(* CODESYS project BaseVista.library
   Company: Vistaprint
   Title: Base_PLC
   Description: 0.3.5.10	- delete cmd on OFF/EOFF alarm
      	- delete SubState on state change
      	- alarm children propagation set true
      0.3.5.9	- goes to OFFBusy from EOFF
      	- added FurtherReactions to Always
      0.3.5.8 	- Added disable Child Alarm propagation functionality
      0.3.5.7 	- Added two actions to disable the EOFF and OFF Alarm transition
      0.3.5.6 	- fixed ERRORQuit
      0.3.5.5 	- TwinCAT 3.1 4016.12
      	- Added a Simulate all to the CIf.Info. This propagates the simulation comand down
      	- Added disable variables to the me for the EOff & Off Alarm and Comand
      	- Added new versions of Tc2_System & Tc2_Utilities
      0.3.5.4 	- added Full Name to CIf
      0.3.5.3 	- Compiled with 3.1 4016.6
      	- Added InstancePath to CIf.Info
      	- Added a property for InstancePath
      	- Fill CIf.Info.InstancePath in FB_init
      0.3.5.2 - CtrlInit() uses internal variable again, in cyclic call of FB at first caclic call and init not done - only init is executed
      	- Alarmhandler works now with time stamp FB, properties for timestamp usage in controller
      	- Add new functions strstr, initAllCtrl, callAllCtrlInit
      	- Integrate in BaseCtrl state logging
      	- Add logger system
      - Add time stamp FUB FB_TimeStamp
      0.3.5.1 - Add Methode ResetSubState
      - alarm reset first statemachine and then the messages
      0.3.5.0 - Update to TwinCat 4016.5
      0.3.4.9 - Increased maxchildnumber to 30
                  - CtrlInit made Public
                  - New CtrlInit call only once flag
      0.3.4.8 - BugFix setAlarm (rst,clr & set)
      0.3.4.7 - Increased the maxchildnumber to 25
      0.3.4.6 - Increased the maxchildnumber to 40
      0.3.4.5 - BugFix in alarm manager
      0.3.4.2 - Changed the Pramas Text in FB_CtrlBase
      0.3.4.1 - State single answer. Reset pending alarm class to NONE.
      0.3.4.0 - New CheckAllChildState also true feedback if check state of child OFF or EOFF and child in ERROR;
      - Bug fix Always Single-answer and startup with wait on PON
      - FB_Alm_Man: New Property IsInitDone		feedback at least one valid time stamp read out 
      0.3.3.7 - CheckParentAlmClass OFF and STOP added -> reaction of Controller
      0.3.3.6 - FB_Alm_Man Property CntPerClass added, alarm classes EOFF, OFF and STOP from parent to child, in EOFFBusy and OFF busy command in cyclic action (not entry action)
      
      0.3.3.4 - Added IO support for USINT datatype
      
      0.3.3.3 - Bug fixed in getInBolDebounced(FUN)
      
      0.3.3.2 - New function setAllCtrlAlarmFB -> all controller init pointer of alarmhandler; 
      - Rename GetInUint ->getInUint; 
      - New function ScaleINT (scale integer variable p.e. analog increment to 0.1mm)
      
      0.3.3.1  Added getInBolDebounced(FUN) and T_Ctrl_IoBoolDebounced(STRUCT) for debouncing inputs
      0.3.3.0 - Added pfbAlarmCtrl and the "zugehörige" property to allow clean alarm calls also from controllers in libraries.
      0.3.2.0 - Del getCtrlCIF,iniCtrlArray; Set cmds to child EOFF,OFF,PON; EOFF State; Check child ALM EOFF     
      0.3.1.3 - Bugfix
      0.3.1.2 - Added iniAllCtrlArrays - this is iniCtrlArray + the cif array
      0.3.1 - Added the automatic EOff propagation.
      0.3.0 - Added the substate to T_CTRL_CLASS_STATEMACHINE
      Automatic Substate handling.
      0.2.3 - Added support for sub usec cycletimes
      0.2.2 - Added the UInt for IO. T_CTRL_IOUint, setInUint(), setOutUint()
      0.2.1 - Added the property CtrlCIf to FB_CtrlBase
   Version: 0.3.5.10

Project tree, tasks and I/O mapping:
  libraries: Tc2_Standard, 3.3.0.0 (Beckhoff Automation GmbH); Tc2_System, 3.3.8.1 (Beckhoff Automation GmbH); Tc2_Utilities, 3.3.8.0 (Beckhoff Automation GmbH); Tc3_Interfaces, 3.3.0.0 (Beckhoff Automation GmbH); Tc3_MemMan, 3.3.1.0 (Beckhoff Automation GmbH); Tc3_Module, 3.3.6.0 (Beckhoff Automation GmbH)
  POUs/
    Alarm/
      data type E_AlmClass
      data type E_AlmCmd
      data type E_AlmState
      function block FB_Alm_Man [ST]: aCntPerClass, clearAlarm, IsInitDone, LocalTime_FileTime_BaseWin, LocalTime_TimeStruct_BaseWin, setAlarm, UTC_FileTime, UTC_TimeStruct
      data type T_AlmElement
      data type T_Ctrl_Alm
    BaseCtrl/
      global variables Base_CmdState
      global variables Base_Const
      data type E_Mode
      function block FB_CtrlBase [ST]: AddChild, AlarmCtrl, Always, BaseLog, CheckAllChildAlmClass, CheckAllChildState, CheckChildAlmClass, CheckCmdValid, CheckParentAlmClass, ChildrenAlarmPropagation, ClearAllSimulation, CtrlCIf, CtrlFB, CtrlInit, CycleEndDuty, CycleStartDuty, EOFF_EntryAction, EOffAlarmTransition, FB_init, FurtherReactions, getCmdState, iniAllCtrlArrays, InstancePath, IoInBridge, IoOutBridge, OffAlarmTransition, ResetSubState, SetAllChildAlmClass, SetAllChildCmd, SetAllSimulation, sta_EOFF, sta_EOFFBusy, sta_ERROR, sta_ERRORQuit, sta_OFF, sta_OFFBusy, sta_PON, sta_PONBusy, sta_SINGLE_ANSWER, StateMachine
      interface I_CtrlBase: CtrlCIf, CtrlFB
      data type T_Ctrl_AlarmConfig
      data type T_Ctrl_CIf
      data type T_Ctrl_Class
      data type T_Ctrl_Class_Alm
      data type T_Ctrl_Class_StateMachine
      data type T_Ctrl_CmdListElement
      data type T_Ctrl_Info
      data type T_Ctrl_IoBool
      data type T_Ctrl_IoBoolDebounced
      data type T_Ctrl_IoInt
      data type T_Ctrl_IoUint
      data type T_Ctrl_IoUsint
      data type T_Ctrl_Job
      data type T_Ctrl_SwCfg
      data type T_fbInfo
      data type T_StateLogger
    Utility/
      DLL (Double Linked List)/
        function block FB_DLL [ST]: addElement, deleteAll, deleteElement, FB_init, firstElement, numberOfElements, searchElement
        data type T_Element
      FileFolder/
        function block FB_FileCopy [ST]
        function block FB_FileHdl [ST]: ActFileSize, M_Cmd_FileDelete, M_Cmd_NewFile, M_Cmd_WriteBuffer, M_FileClose, M_FileCopy, M_FileDelete, M_FileOpen, M_FileRename, M_FileWrite, M_GetPathName, M_Init
        function block FB_FolderHdl [ST]: FileSupervisionPeriod, get_FileList, get_NewestFileEntry, M_Cmd_RefreshFileList, M_FileDelete, M_FileExist, M_getFileInfo, M_GetFileSize, M_Init, M_RefreshFileList, M_SortFileList, MaxNrOfFilesInFolder
        global variables FileHdl
      Logger/
        BasLog/
          global variables BasLog
          function block FB_BasLog [ST]: M_ChangeMask, M_CheckValidLogType, M_ClientInit, M_GetHandle, M_Log, M_Read
          function block FB_BasLogTest_Client [ST]
          function block FB_BasLogTest_Sender [ST]
          data type T_Bl_BaseStruc
          data type T_Bl_LibClient
          data type T_Bl_LibHandleRow
          data type T_Bl_LibSingleClient
        DatLog/
          global variables DatLog
          function block FB_DatLog [ST]: M_AllocMEM, M_CheckAndAppendDatLogInfo, M_GetHandle, M_Init, M_Log
          function block FB_DatLogTest_Sender [ST]
          data type T_DatLogTest
          data type T_DL_Item
          data type T_DL_LibInfo
          data type T_DL_Statemachine
          data type T_DL_SysInfo
        FileLc/
          function block FB_FileLc [ST]: M_Cyclic, M_Init, M_PutPvIdInList, M_ReleaseBuffer, M_WriteActItemIdx, M_WriteRecord
          function block FB_FileLc_FileHdl [ST]: ActFileSize, M_Cyclic, M_Init
          function block FB_FileLc_WorkOnFile [ST]: FB_exit, M_AllocMEM, M_ReleaseAllMEM
          function block FB_FileLcTest [ST]
          global variables FileLc
          data type T_FileLc_FileHandler
          data type T_FileLc_ItemCfg
          data type T_FileLc_ItemData
          data type T_FileLc_ItemInfo
          data type T_FileLc_LibInfo
          data type T_FileLc_RecordData
          data type T_FileLc_Statemachine
          data type T_FileLc_SysCfg
          data type T_FileLc_SysDebugInfo
          data type T_FileLc_SysInfo
      Queue/
        function block FB_Queue [ST]: FB_exit, M_AllocNewQueue, M_AllocNewQueueInfo, M_AllocNewQueueSystem, M_CheckAndAppendQueueSysInfo, M_Clear, M_GetHandle, M_GetHandle_TC, M_Init, M_Read, M_ReadReference, M_Write
        function block FB_QueueTest_Receiver [ST]
        function block FB_QueueTest_Sender [ST]
        global variables Queue
        data type T_Queue_Info
        data type T_Queue_InfoInternal
        data type T_Queue_LibInfo
        data type T_Queue_SysDebugInfo
        data type T_Queue_SysInfo
        data type T_Queue_TestData
      function callAllCtrlInit [ST]
      function block FB_TimeStamp [ST]: LocalTime_FileTime_BaseUTC, LocalTime_FileTime_BaseWin, LocalTime_TimeStruct_BaseUTC, LocalTime_TimeStruct_BaseWin, TimeZone_Refresh, UTC_FileTime, UTC_TimeStruct
      function getInBol [ST]
      function getInBolDebounced [ST]
      function getInInt [ST]
      function getInUint [ST]
      function getInUsint [ST]
      function getStrInstanceName [ST]
      function initAllCtrl [ST]
      function ScaleINT [ST]
      function setAllCtrlAlarmFB [ST]
      function setAllCtrlBasLogFB [ST]
      function setOutBol [ST]
      function setOutInt [ST]
      function setOutUint [ST]
      function setOutUsint [ST]
      function strstr [ST]
  Version/
    global variables Global_Version
*)

// POUs/Alarm/E_AlmClass
/// Do not change the sequence in this struct, such that the highest number is always the most important alarm!
TYPE E_AlmClass :
(
	///no alarm active
	NONE := 0,
	///info
	INFO,
	///warning
	WARNING,
	///tact stop
	TSTOP,
	///stop
	STOP,
	///off
	OFF,
	///Emergency off
	EOFF,
	Max_E_AlmClass
) INT;
END_TYPE

// POUs/Alarm/E_AlmCmd
TYPE E_AlmCmd :
(
	DONE := -1,
	INITIALIZED := 0,
	RESET_ALL := 2,
	RESET_RST := 4,
	RESET_CLR := 6,
	Max_E_AlmCmd
);
END_TYPE

// POUs/Alarm/E_AlmState
TYPE E_AlmState :
(
	///no alarm active
	NONE := 0,
	///alarm clear entry -> set bit1
	CLR := 1,
	///entry resettable alarm ->  set bit2
	RST := 2,
	///entry non resettable alarm ->  set bit2 + bit3
	SET := 3,
	Max_E_AlmState
);
END_TYPE

// POUs/Alarm/T_AlmElement
TYPE T_AlmElement :
STRUCT
	///unique alarm number := 100000*udiMachineNr + intCtrlId*100 + udiAlarmNr
	udiNr: UDINT;
	///additional information - better string???
	dinInfo: DINT;
	///corresponding alarm class
	eClass: E_AlmClass;
	///clear, resetable
	intState: E_AlmState;
	///entry time
	strDTEntry: STRING;
	///from machine (standard = 1)
	udiMachineNr: UDINT;
	///from controller
	intCtrlId: INT;
	///local alarm number
	udiAlarmNr: UDINT;
	// for debugging string alarm controller-alarm
	strText: STRING;
END_STRUCT
END_TYPE

// POUs/Alarm/T_Ctrl_Alm
TYPE T_Ctrl_Alm :
STRUCT
	///alarm flag array
	bol: BOOL;
	eAlmClass: E_AlmClass;
	strText: STRING;
END_STRUCT
END_TYPE

// POUs/BaseCtrl/E_Mode
{attribute 'qualified_only' := ''}
TYPE E_Mode :
(
	INITIALIZED := 0,
	AUTO := 10,
	SEMI := 11,
	MANU := 12
) INT;
END_TYPE

// POUs/BaseCtrl/T_Ctrl_AlarmConfig
TYPE T_Ctrl_AlarmConfig :
STRUCT
	// Disable the OFF Alarm transition
	bolOffAlarmTransitionDisable	: BOOL;
	// Disable the EOFF Alarm Transition
	bolEOffAlarmTransitionDisable	: BOOL;
	// Disable to Off Command Transition 
	bolOffCmdTransitionDisable		: BOOL;
	// Disable the EOffCommandTransition
	bolEOffCmdTransitionDisable		: BOOL;
	// Enable Alarm Propagation to Children
	bolChildrenAlarmPropagation		: BOOL;
END_STRUCT
END_TYPE

// POUs/BaseCtrl/T_Ctrl_CIf
TYPE T_Ctrl_CIf :
STRUCT
	Job: T_Ctrl_Job;
	Info: T_Ctrl_Info;
	SwCfg: T_Ctrl_SwCfg;
END_STRUCT
END_TYPE

// POUs/BaseCtrl/T_Ctrl_Class
TYPE T_Ctrl_Class :
STRUCT
	///local test flag to supress cyclic run (for debugging after init)
	bolActivate					: BOOL;
	intCmd						: INT;
	intCmdLast					: INT;
	eModeHistory				: E_Mode;
	///local flag mode change detected
	bolChangeBackToAUTO			: BOOL;
	StateMachine				: T_Ctrl_Class_StateMachine;
	SubStateMachine				: T_Ctrl_Class_StateMachine;
	Alarm						: T_Ctrl_Class_Alm;
	FUBInfo						: T_fbInfo;
	AlarmConfig					: T_Ctrl_AlarmConfig;
	// StateLogger infos
	stStateLogger : T_StateLogger;
	// Simulate All Executed
	bolSimulateAllExecuted			: BOOL;
END_STRUCT
END_TYPE

// POUs/BaseCtrl/T_Ctrl_Class_Alm
TYPE T_Ctrl_Class_Alm :
STRUCT
	bolResetOk: BOOL;
	///flag positive check me alarm from child
	bolfp: BOOL;
	///local activ alarm class of parent ctrl
	eParent_ActivAlmClass: E_AlmClass;
	///highest local activ alarm class
	eActivAlmClass: E_AlmClass;
END_STRUCT
END_TYPE

// POUs/BaseCtrl/T_Ctrl_Class_StateMachine
TYPE T_Ctrl_Class_StateMachine :
STRUCT
	///actual state
	intState: INT;
	///state of last cycle
	intStateLastCycle: INT;
	///save history backup p.e. in ERROR state
	intStateHistory: INT;
	///set state for next cycle
	intStateNext: INT;
	///[ms] to simulate state in SINGLE_ANSWER
	udiStateSimSetTime_ms: UDINT := 1000;
	///[ms] time in one state
	udiTimeInState_ms: UDINT;
	///[ms] time in one state
	relTimeInState_ms: REAL;
	///[us] time in one state
	udiTimeInState_us: UDINT;
END_STRUCT
END_TYPE

// POUs/BaseCtrl/T_Ctrl_CmdListElement
TYPE T_Ctrl_CmdListElement :
STRUCT
	///command implemented in controller
	intCmd: INT;
	///command is available info for UI
	bolAvailable: BOOL;
	/// Name of command. Important for UI.
	strName: STRING(80);
END_STRUCT
END_TYPE

// POUs/BaseCtrl/T_Ctrl_Info
TYPE T_Ctrl_Info :
STRUCT
	///name of controller instance
	strName				: STRING(80);
	///full name of controller instance
	strFullName			: STRING(80);
	///class of controller
	strType				: STRING(80);
	///unique controller instance identification number
	intCtrlId			: INT;
	///unique identification number of parent controller instance
	intParentCtrlId		: INT;
	///all inputs valid -> init done
	bolInitDone			: BOOL;
	///Childs
	p_afbChild			: ARRAY[0..Base_Const.cMaxNrOfChilds] OF POINTER TO FB_CtrlBase;
	///common interface array of childs
	p_aCIf				: ARRAY[0..Base_Const.cMaxNrOfChilds] OF POINTER TO T_Ctrl_CIf;
	// Child Count
	uinChildNbr			: UINT;
	// Absolut path to the controller
	strInstancePath		: STRING;
END_STRUCT
END_TYPE

// POUs/BaseCtrl/T_Ctrl_IoBool
TYPE T_Ctrl_IoBool :
STRUCT
	///mapped io variable to hardware
	map: BOOL;
	///shows the state of (input: mapped, output: set by programm respectiv at the moment one cycle later evtl. from the forcing if forcing active) -> necessary for what?
	state: BOOL;
	///variabel to/ from program
	intern: BOOL;
	///variabel set from UI
	force: BOOL;
	///enable force of single io-datapoint
	EnForce: BOOL;
END_STRUCT
END_TYPE

// POUs/BaseCtrl/T_Ctrl_IoBoolDebounced
TYPE T_Ctrl_IoBoolDebounced :
STRUCT
	///mapped io variable to hardware
	map: BOOL;
	///shows the state of (input: mapped, output: set by programm respectiv at the moment one cycle later evtl. from the forcing if forcing active) -> necessary for what?
	state: BOOL;
	///variabel to/ from program
	intern: BOOL;
	///variabel set from UI
	force: BOOL;
	///enable force of single io-datapoint
	EnForce: BOOL;
	// time since last input change
	udinDebouncedTimeCounter_ms: UDINT;
END_STRUCT
END_TYPE

// POUs/BaseCtrl/T_Ctrl_IoInt
TYPE T_Ctrl_IoInt :
STRUCT
	///mapped io variable to hardware
	map: INT;
	///shows the state of (input: mapped, output: set by programm respectiv at the moment one cycle later evtl. from the forcing if forcing active) -> necessary for what?
	state: INT;
	///variabel to/ from program
	intern: INT;
	///variabel set from UI
	force: INT;
	///enable force of single io-datapoint
	EnForce: BOOL;
END_STRUCT
END_TYPE

// POUs/BaseCtrl/T_Ctrl_IoUint
TYPE T_Ctrl_IoUint :
STRUCT
	///mapped io variable to hardware
	map: UINT;
	///shows the state of (input: mapped, output: set by programm respectiv at the moment one cycle later evtl. from the forcing if forcing active) -> necessary for what?
	state: UINT;
	///variabel to/ from program
	intern: UINT;
	///variabel set from UI
	force: UINT;
	///enable force of single io-datapoint
	EnForce: BOOL;
END_STRUCT
END_TYPE

// POUs/BaseCtrl/T_Ctrl_IoUsint
TYPE T_Ctrl_IoUsint :
STRUCT
	///mapped io variable to hardware
	map: USINT;
	///shows the state of (input: mapped, output: set by programm respectiv at the moment one cycle later evtl. from the forcing if forcing active) -> necessary for what?
	state: USINT;
	///variabel to/ from program
	intern: USINT;
	///variabel set from UI
	force: USINT;
	///enable force of single io-datapoint
	EnForce: BOOL;
END_STRUCT
END_TYPE

// POUs/BaseCtrl/T_Ctrl_Job
TYPE T_Ctrl_Job :
STRUCT
	///mode if mode = AUTO -> ACmd will be used, otherwise the MCmd channel is open
	eMode: E_Mode;
	///automatic command from parent ctrl
	intACmd: INT;
	///manual command from UI p.e.
	intMCmd: INT;
	///active cmd
	strCmd: STRING;
	///active state
	intState: INT;
	strState: STRING;
	///if used - show substates for debugging
	strSubState: STRING;
	///event channel to signal special events to parent parallel to status
	intEvt: INT;
	///reset all alarms
	bolAlmReset: BOOL;
	///activate io-forcing
	bolIoForce: BOOL;
	///overwrite suspend all interlocks (for debugging/testing)
	bolIlkOverwrite: BOOL;
	///activ alarm class of parent ctrl
	eParent_ActivAlmClass: E_AlmClass;
	///activ alarm class of me ctrl
	eMe_ActivAlmClass: E_AlmClass;
	///list of all implemented commands
	aCmdList: ARRAY[0..cMaxCmdPerCtrl] OF T_Ctrl_CmdListElement;
END_STRUCT
END_TYPE

// POUs/BaseCtrl/T_Ctrl_SwCfg
TYPE T_Ctrl_SwCfg :
	STRUCT
		///hardware/controller exists
		bolExist: BOOL;
		///enable statemachine
		bolEnable: BOOL;
		///set controller in simulation(statemachine active, io local simulated)
		bolSimulation: BOOL;
		//set controller and all sub controllers into simulation(statemachine active, io local simulated)
		bolAllSimulation: BOOL;
		// enable statelogger
		bolEnStateLogger: BOOL;
	END_STRUCT
END_TYPE

// POUs/BaseCtrl/T_fbInfo
TYPE T_fbInfo :
STRUCT
	bolCycleTimeBelowMS			: BOOL;
	udiSample_ms				: UDINT;
	udiSample_us				: UDINT;
END_STRUCT
END_TYPE

// POUs/BaseCtrl/T_StateLogger
TYPE T_StateLogger :
STRUCT
	pfbBaseLog : POINTER TO FB_BasLog; // should be set from outside over property
	uinStatus_Handle : UINT; // =0 handle ok or not allready requested 
	pHandle : POINTER TO T_Bl_LibHandleRow; // pointer to base logger system
	uinStatusWrite : UDINT; // feedback if write was successfully
	bolDoLog : BOOL; // state change detected or application cmd to log infos
	strText1: STRING(BasLog.cMAX_CHAR_TEXT1); // set in CycleEndDuty
	
	// free usable for application
	strText2: STRING(BasLog.cMAX_CHAR_TEXT2); // free usable from application task for additional debug informations
	dinPar3: DINT;	 // free usable from application task for additional debug informations
	dinPar4: DINT;	 // free usable from application task for additional debug informations
END_STRUCT
END_TYPE

// POUs/Utility/DLL (Double Linked List)/T_Element
{attribute 'enable_dynamic_creation' := ''}
TYPE T_Element :
STRUCT
	pPrevElement: POINTER TO T_Element;
	pData: POINTER TO BYTE;
	uliKey: ULINT;
	pNextElement: POINTER TO T_Element;
END_STRUCT
END_TYPE

// POUs/Utility/Logger/BasLog/T_Bl_BaseStruc
TYPE T_Bl_BaseStruc :
STRUCT
	dtDateTimeEntry: DT; // actual date and time (Date and time.The most significat digit is one second. 32Bit 1970-01-01-00:00 to 2106-02-06-06:28:15)
	uinMs : UINT; // actual millisecond
	udiLogType: UDINT; // kind of log
	intCtrlID: INT; // unique controllerID which element has created this entry
	strText1: STRING(BasLog.cMAX_CHAR_TEXT1);	//informationtext1
	strText2: STRING(BasLog.cMAX_CHAR_TEXT2); // informationtext2
	dinPar1: DINT; // value parmeter 1
	dinPar2: DINT; // value parmeter 2
	dinPar3: DINT; // value parmeter 3
	dinPar4: DINT; // value parmeter 4
END_STRUCT
END_TYPE

// POUs/Utility/Logger/BasLog/T_Bl_LibClient
TYPE T_Bl_LibClient :
STRUCT
	stClient : ARRAY [0..BasLog.cMAX_CLIENTS] OF T_Bl_LibSingleClient; // informationstruct for one client
	usiClientNr : USINT; // number of declared clients
	stHandleRow : ARRAY[0..Queue.cMAX_NR_OF_TASKS]OF T_Bl_LibHandleRow; // handle for access Buffer
	p_fbTimeStamp: POINTER TO FB_TimeStamp; // pointer to FB_TimeStamp 
END_STRUCT
END_TYPE

// POUs/Utility/Logger/BasLog/T_Bl_LibHandleRow
TYPE T_Bl_LibHandleRow :
STRUCT
	pQueueHandle :ARRAY[0..BasLog.cMAX_CLIENTS] OF POINTER TO T_Queue_Info; // handle for access buffer
	usiRequest: USINT; // information if task allready requested a handle
END_STRUCT
END_TYPE

// POUs/Utility/Logger/BasLog/T_Bl_LibSingleClient
TYPE T_Bl_LibSingleClient :
STRUCT
	strName : STRING(Queue.cMAX_NAME_LENGTH); // name of declared client
	udiMask : UDINT; // filter mask for selection
	udiNrOfElements: UDINT; // number of elements
	bolUseLocalTimeStamp : BOOL; // definition if using local time or UTC
END_STRUCT
END_TYPE

// POUs/Utility/Logger/DatLog/T_DatLogTest
TYPE T_DatLogTest :
STRUCT
	bolOk : BOOL := TRUE;
	intCnt : INT := 77;
	strNewText : STRING(20) := 'Test Data log';
END_STRUCT
END_TYPE

// POUs/Utility/Logger/DatLog/T_DL_Item
TYPE T_DL_Item :
STRUCT
	strPvName : T_MaxString; // name of declared client
	udiItemType : UDINT; // datatyp defined in logsystem
	uinItemOffset : UINT; // data offset in record struct
	SymInfo : SYMINFOSTRUCT;
END_STRUCT
END_TYPE

// POUs/Utility/Logger/DatLog/T_DL_LibInfo
TYPE T_DL_LibInfo :
STRUCT
	pstDatLogSysInfo : POINTER TO T_DL_SysInfo; // pointer to DL log system list
	stStatemachine: T_DL_Statemachine;
	udiCommonRecIdx: UDINT; // general record idx (because of mutex problematic has to be increased with 2)
END_STRUCT
END_TYPE

// POUs/Utility/Logger/DatLog/T_DL_Statemachine
TYPE T_DL_Statemachine :
STRUCT
	uinState : UINT; (*Status (Statemachine) des Filehandlers*)
	uinState_old : UINT; (*status old for entry action generation*)
	bolExecute_old : BOOL;
	usiInitDone : USINT; (*Merker für Neustart*)
END_STRUCT
END_TYPE

// POUs/Utility/Logger/DatLog/T_DL_SysInfo
TYPE T_DL_SysInfo :
STRUCT
	strDatLogName : STRING(DatLog.cMAX_SYS_NAME_LENGTH);
	usiInitOk : USINT; // initalisation successfully finished
	uinNbrOfItems : UINT; // number of items
	uinStartId : UINT; // StartId
	pBaseLogHandle : POINTER TO POINTER TO T_Queue_Info; // handle from BaseLog Init
	p_fbBasLog: POINTER TO FB_BasLog;
	pstItems: POINTER TO T_DL_Item; // itemlist
	uinCntReadItems : UINT; // read counte
	uinItemOffset : UINT; // offset calculation
	pstNextDatLogSystem : POINTER TO T_DL_SysInfo;
END_STRUCT
END_TYPE

// POUs/Utility/Logger/FileLc/T_FileLc_FileHandler
TYPE T_FileLc_FileHandler :
STRUCT
	uinState : UINT; (*Status (Statemachine) des Filehandlers*)
	uinState_old : UINT; (*status old for entry action generation*)
	usiCmd : USINT; (*Internes Kommando*)
	usiCmdNewFile : USINT; (*Schliesse aktuelles File ab und erstelle ein neues LogFile*)
	usiInitDone : USINT; (*Merker für Neustart*)
	udiWriteTimer : UDINT; (*Zeit seit letztem File Schreibzyklus*)
	p_bytTmpFileBuffer : POINTER TO BYTE; (*Zeiger auf temporären Filebuffer*)
	udiTmpFileBufferSize : UDINT; (*Grösse des temporären Filebuffers*)
	udiTmpFileBufferOffset : UDINT; (*Schreibzeiger des temporären Filebuffers*)
	udiRecordCnt : UDINT; // actual record count in file
	FB_FileLc_FileHdl : FB_FileLc_FileHdl; // FUB instance
	strInfo: Tc2_System.T_MaxString;	// additional debug Info
END_STRUCT
END_TYPE

// POUs/Utility/Logger/FileLc/T_FileLc_ItemCfg
TYPE T_FileLc_ItemCfg :
STRUCT
	dinPvId : DINT; (*Item - Id*)
	strPostText : STRING[FileLc.cPRE_POST_TEXTLEN]; (*Text, der nach dem Item - Value ins File geschrieben wird.*)
END_STRUCT
END_TYPE

// POUs/Utility/Logger/FileLc/T_FileLc_ItemData
TYPE T_FileLc_ItemData :
STRUCT
		udiRecIdx : UDINT; (*Record - Index, zu welchem die Daten gehören*)
		strValue : STRING[FileLc.cMAX_ITEM_CHAR]; (*Item - Value bereits in einen String gewandelt*)
END_STRUCT
END_TYPE

// POUs/Utility/Logger/FileLc/T_FileLc_ItemInfo
TYPE T_FileLc_ItemInfo :
STRUCT
	uinActNbrOfItems : UINT; (*Anzahl ermittelter Items*)
	strPreItemText : STRING[FileLc.cPRE_POST_TEXTLEN]; (*Text, der vor dem ersten Item - Value ins File geschrieben wird*)
	p_bytItemCfgList : POINTER TO T_FileLc_ItemCfg;; (*Zeiger auf die Item - Konfig - Liste*)
	stItemRecordData : ARRAY[0..Queue.cMAX_NR_OF_TASKS] OF T_FileLc_RecordData; (*Record - Data: Da Data - Records theoretisch unterbrochen werden können (Taskklassenprio), müssen mehrere Records quasi parallel behandelt werden können. Jeder Record hat daher seinen eigenen Index.*)
	a_p_bytItemDataList : ARRAY[0..Queue.cMAX_NR_OF_TASKS] OF POINTER TO BYTE; (*Item - Data: siehe oben...*)
END_STRUCT
END_TYPE

// POUs/Utility/Logger/FileLc/T_FileLc_LibInfo
TYPE T_FileLc_LibInfo :
STRUCT
	uinActNbrOfFileClients: UINT; // number of file clients
	uinActClientInitActive: UINT; // =0 ready for next client, actual active init of client nr
	stSysInfo : ARRAY[0..FileLc.cMAX_NBR_OF_FILECLIENTS] OF T_FileLc_SysInfo;
	p_fbBasLog: POINTER TO FB_BasLog; // only one central FB_BasLog instance allowed per PLC!!!
	fbTimeStamp: FB_TimeStamp; // only one central time for time stamps
END_STRUCT
END_TYPE

// POUs/Utility/Logger/FileLc/T_FileLc_RecordData
TYPE T_FileLc_RecordData :
STRUCT
	udiRecIdx : UDINT; (*Record - Index*)
	dtActDateTime : DATE_AND_TIME; (*Datum/Zeit der Record - Daten*)
	uinActMilli : UINT; (*Millisekunden der Record - Daten*)
END_STRUCT
END_TYPE

// POUs/Utility/Logger/FileLc/T_FileLc_Statemachine
TYPE T_FileLc_Statemachine :
STRUCT
	uinState : UINT; (*Status (Statemachine) des Filehandlers*)
	uinState_old : UINT; (*status old for entry action generation*)
	usiInitDone : USINT; (*Merker für Neustart*)
END_STRUCT
END_TYPE

// POUs/Utility/Logger/FileLc/T_FileLc_SysCfg
TYPE T_FileLc_SysCfg :
STRUCT
	uinMaxNbrOfLogFiles : UINT; (*Maximale Anzahl Log-Files*)
	udiTimeCheckMaxFileNr :UDINT; // [ms] time until check if more then max number of files exist in folder -> delete oldest
	uinNewFileOnRestart : UINT; (*Nach Steuerungsneustart neues File anlegen, wenn Wert > 0*)
	udiMaxTimeWriteToFile : UDINT; (*Maximale Zeit zwischen zwei File - Schreibzyklen*)
	bolUseLocalTimeStamp : BOOL; // define if using local time or UTC
	strLogFileNameExt : STRING[FileLc.cFILENAME_LENGTH]; (*Extension des Logfiles*)
	strLogFileNamePraeFix : STRING[FileLc.cFILENAME_LENGTH]; (*Präfix des Logfiles*)
	strLogPath : STRING[FileLc.cFILENAME_LENGTH]; (*Verzeichnis in welchem die Logfiles angelegt werden*)
	strLogNetId : STRING(23); // to access foreign system drives where TinCat has to be installed!!! Is a string containing the AMS network identifier of the target device to which the ADS command is directed.
	udiQueueLen : UDINT; (*Queue Länge der BaseLog - Queue*)
	udiMaxFileSize : UDINT; (*Maximale Dateigrösse eines Logfiles*)
	udiMaxEntriesInFile : UDINT; (*Maximale Anzahl Einträge in einem Logfile*)
END_STRUCT
END_TYPE

// POUs/Utility/Logger/FileLc/T_FileLc_SysDebugInfo
TYPE T_FileLc_SysDebugInfo :
STRUCT
		udiLogCounter : UDINT;
		uinGetHandleCalls : UINT;
END_STRUCT
END_TYPE

// POUs/Utility/Logger/FileLc/T_FileLc_SysInfo
TYPE T_FileLc_SysInfo :
STRUCT
	strPathName : STRING[FileLc.cPATH_LENGTH]; (*device name for config - file*)
	pBaseLogHandle : POINTER TO POINTER TO T_Queue_Info; // handle from BaseLog Init
	uinLogTyp : UINT; (* LogTyp*)
	udiMask : UDINT; (*actual log mask*)
	udiCylceTimeMs : UDINT; (*cycle time in milli seconds*)
	p_bytHeaderText : POINTER TO BYTE; (*Zeiger auf den Header Text*)
	udiHeaderTextLen : UDINT; (*Footer text len*)
	p_bytFooterText : POINTER TO BYTE; (*Zeiger auf den Footer Text*)
	udiFooterTextLen : UDINT; (*Footer text len*)
	p_bytTmpRecordText : POINTER TO BYTE; (*Zeiger auf den temporären Record - Text*)
	udiTmpRecordSize : UDINT; (*Grösse des temporären Record - Text*)
	udiTmpRecordLen : UDINT; (*Aktuelle Länge des temporären Record - Text*)
	bolTmpRecordFull : BOOL; (*temp record is full - text is full --> do write in file buffer*)
	stConfig : T_FileLc_SysCfg; (*config data*)
	stFileHandler : T_FileLc_FileHandler; (*Filehandler*)
	stItemInfo : T_FileLc_ItemInfo; (*Item-Infos --> <RECORD> Items.... </RECORD>*)
	stStatemachine : T_FileLc_Statemachine;
	fbFileLc_WorkOnFile : FB_FileLc_WorkOnFile;
END_STRUCT
END_TYPE

// POUs/Utility/Queue/T_Queue_Info
{attribute 'enable_dynamic_creation' := ''}
TYPE T_Queue_Info :
STRUCT
	fbBuffer: FB_MemRingBuffer; // Buffer FB
	udiFillLevel : UDINT; // % actual used buffer size
	pQueueSysInfo: POINTER TO T_Queue_SysInfo; // pointer to sytem struct (parent)
	bolAllocMe:BOOL; //flag gethandle called before init done!!!
END_STRUCT
END_TYPE

// POUs/Utility/Queue/T_Queue_InfoInternal
TYPE T_Queue_InfoInternal :
STRUCT
	bolAllocated:BOOL; //queue allocated
	fbBuffer: FB_MemRingBuffer; // Buffer FB
	udiFillLevel : UDINT; // % actual used buffer size
END_STRUCT
END_TYPE

// POUs/Utility/Queue/T_Queue_LibInfo
TYPE T_Queue_LibInfo :
STRUCT
	pstQueue_SysInfo : POINTER TO T_Queue_SysInfo; // pointer to first queue system - linked list 
	uinFUBInternalError: UINT; // internal error
	stSysDebugInfo:T_Queue_SysDebugInfo; //Debug structure
END_STRUCT
END_TYPE

// POUs/Utility/Queue/T_Queue_SysDebugInfo
TYPE T_Queue_SysDebugInfo :
STRUCT
	uinGetHandleCalls : UINT;
	uinIniCalls:UINT;
	uinCheckAndAppendQSCalls:UINT;
	uinAllocNewQSCalls: UINT;
	uinAllocNewQICalls: UINT;
	uinAllocnewQCalls:UINT;
END_STRUCT
END_TYPE

// POUs/Utility/Queue/T_Queue_SysInfo
{attribute 'enable_dynamic_creation' := ''}
TYPE T_Queue_SysInfo :
STRUCT
	strQueueName : STRING(Queue.cMAX_NAME_LENGTH); // queue name
	uinNbrOfElement : UINT; // number of elements
	udiSizeOfElement : UDINT; // Byte size of one elment
	uinMode : UINT; // 0: FIFO ring buffer, no overwrite!!
	// ident of FIFO new saved in fbBuffer udiIdent : UDINT;
	udiSecure: UDINT; // alternating bit muster for plausibility check of handle
	pQueueInfo: ARRAY[0..Queue.cMAX_NR_OF_TASKS] OF POINTER TO  T_Queue_Info; // structure/queue per tasclass
	pstNextQueue_SysInfo : POINTER TO T_Queue_SysInfo; // pointer to next queue system - linked list 
END_STRUCT
END_TYPE

// POUs/Utility/Queue/T_Queue_TestData
TYPE T_Queue_TestData :
STRUCT
	strName : STRING(34); //name OF process variabel
	usiDataTyp : USINT;
	udiDataLen : UDINT;
	udiDimension : UDINT;
	udiAdress : UDINT;
END_STRUCT
END_TYPE

// POUs/BaseCtrl/Base_CmdState
VAR_GLOBAL CONSTANT
	///ctrl commands definitions
	///general commands 2-200 - every command has to be a even number
	cCMD_DONE: INT := -1;
	cCMD_INITIALIZED: INT := 0;
	cCMD_PON: INT := 2;
	cCMD_EOFF: INT := 4;
	cCMD_OFF: INT := 6;
	cCMD_INIT: INT := 8;
	cCMD_RUN: INT := 10;
	cCMD_STOP: INT := 12;
	cCMD_TSTOP: INT := 14;
	///ctrl states definitions
	cSTA_DONE: INT := cCMD_DONE;
	cSTA_INITIALIZED: INT := cCMD_INITIALIZED;
	cSTA_PONBusy: INT := 1;
	cSTA_PON: INT := cCMD_PON;
	cSTA_EOFFBusy: INT := 3;
	cSTA_EOFF: INT := cCMD_EOFF;
	cSTA_OFFBusy: INT := 5;
	cSTA_OFF: INT := cCMD_OFF;
	cSTA_INITBusy: INT := 7;
	cSTA_INIT: INT := cCMD_INIT;
	cSTA_RUNBusy: INT := 9;
	cSTA_RUN: INT := cCMD_RUN;
	cSTA_STOPBusy: INT := 11;
	cSTA_STOP: INT := cCMD_STOP;
	cSTA_TSTOPBusy: INT := 13;
	cSTA_TSTOP: INT := cCMD_TSTOP;
	///special states without corresponding cmd
	cSTA_ERROR: INT := 150;
	cSTA_ERRORQuit: INT := 151;
	cSTA_SINGLE_ANSWER: INT := 152;
END_VAR

// POUs/BaseCtrl/Base_Const
VAR_GLOBAL CONSTANT
	///number of child access possible in one controller class
	cMaxNrOfChilds: UINT := 30;
	///maximal number of commands implemented in one controller class
	cMaxCmdPerCtrl: UINT := 15;
	///maximal number of commands implemented in one controller class
	cMaxBaseCmdState: UINT := 200;
END_VAR

// POUs/Utility/FileFolder/FileHdl
VAR_GLOBAL CONSTANT
	cFILE_HDL_MAX_NR_OF_FILE_TO_MANAGE: UDINT := 500;
END_VAR

// POUs/Utility/Logger/BasLog/BasLog
VAR_GLOBAL CONSTANT
	// internal
	cCLIENT_NAME_PF : STRING(10) := '__logClnt'; //Prefix for client name
	cVAR_TYPE_CMD_NEW_REC : USINT := 201; // command for log-records (collect multiple base log entries)
	cVAR_TYPE_CMD_END_REC : USINT := 202; // command for log-records (collect multiple base log entries)
	
	// limits
	cMAX_CLIENTS : USINT := 5; // maximal number of clients 
	cMAX_CHAR_TEXT1: USINT := 80;	// maximal number of chars for information text1
	cMAX_CHAR_TEXT2: USINT := 80;	// maximal number of chars for information text2	
	
	// log types
	cLOGTYPE_ALARM : UDINT:=1; //logtyp alarm
	cLOGTYPE_WARNING : UDINT:=2; //logtyp warning
	cLOGTYPE_INFO : UDINT:=4; //logtyp info
	cLOGTYPE_STATELOG : UDINT:=8; //logtyp state log (for statmachine diagnostic)
	cLOGTYPE_PV_EVENT : UDINT:=16; //logtyp triggered value log
	cLOGTYPE_PV_CYCLIC : UDINT:=32; //logtyp cyclic value log 
	cLOGTYPE_DATA : UDINT:=64; //logtyp data logger
	
	// error number
	cERR_TOO_MANY_CLIENTS : UINT := 51001; // max number of clients connected
	cERR_SYSTEM_NOT_FOUND : UINT := 51002; // the system with this name does not exist
	cERR_INVALID_LOGTYPE : UINT := 51003; // log type is not correct bit coded
	cERR_NO_WRITE_TASK : UINT := 51004; // no client added (no handle from a task)
	cERR_NO_HANDLE : UINT := 51005; // no handle received => fbGetHandle()
	cERR_NO_FB_TIME_STAMP_POINTER : UINT := 51006; // no pointer for FB_TimeStamp
	cERR_NO_FB_TIME_STAMP_INIT_NOT_OK : UINT := 51007; // time stamp value not ready for read out
END_VAR

// POUs/Utility/Logger/DatLog/DatLog
VAR_GLOBAL CONSTANT
	// internal
	cVAR_TYPE_BOOL : USINT := 1; (*Variable hat den Datentyp BOOL*)
	cVAR_TYPE_SINT : USINT := 2; (*Variable hat den Datentyp SINT*)
	cVAR_TYPE_INT : USINT := 3; (*Variable hat den Datentyp INT*)
	cVAR_TYPE_DINT : USINT := 4; (*Variable hat den Datentyp DINT*)
	cVAR_TYPE_USINT : USINT := 5; (*Variable hat den Datentyp USINT*)
	cVAR_TYPE_UINT : USINT := 6; (*Variable hat den Datentyp UINT*)
	cVAR_TYPE_UDINT : USINT := 7; (*Variable hat den Datentyp UDINT*)
	cVAR_TYPE_LREAL : USINT := 10; (*Variable hat den Datentyp REAL*)
	cVAR_TYPE_REAL : USINT := 8; (*Variable hat den Datentyp REAL*)
	cVAR_TYPE_STRING : USINT := 9; (*Variable hat den Datentyp STRING*)
	cVAR_TYPE_DATE_AND_TIME : USINT := 11; (*Variable hat den Datentyp DATE_AND_TIME*)
	cCTRL_ID : INT := 32001; // control ID from data log

	// limits	
	cMAX_SYS_NAME_LENGTH : USINT := 30; //max name length of system data log name
	cMAX_VAR_NAME_LEN : USINT := 50; // max len of variable name
	cMAX_NR_OF_VAR : UINT := 20; // max number of variables definable to log

	// error number	
	cERR_MEM_ALLOC : UINT := 53001; // error on allocating memory 
	cERR_NO_HANDLE : UINT := 53002; // no handle received => fbGetHandle()
	cERR_NO_DATE : UINT := 53003; // no valid data pointer received
	cERR_INIT_FAILED : UINT := 53006; // 
	cERR_NO_ITEMS : UINT := 53004; // 
	cERR_UNSUPPORTED_TYPE : UINT := 53005; // the system support this datatyp not
	cERR_UNSUPPORTED_TYPE_STRING_TOO_LONG : UINT := 53006; // defined string in base log shorter then log string
END_VAR

// POUs/Utility/Logger/FileLc/FileLc
VAR_GLOBAL CONSTANT
	// internal
	cVAR_TYPE_BOOL : USINT := 1; (*Variable hat den Datentyp BOOL*)
	cVAR_TYPE_SINT : USINT := 2; (*Variable hat den Datentyp SINT*)
	cVAR_TYPE_INT : USINT := 3; (*Variable hat den Datentyp INT*)
	cVAR_TYPE_DINT : USINT := 4; (*Variable hat den Datentyp DINT*)
	cVAR_TYPE_USINT : USINT := 5; (*Variable hat den Datentyp USINT*)
	cVAR_TYPE_UINT : USINT := 6; (*Variable hat den Datentyp UINT*)
	cVAR_TYPE_UDINT : USINT := 7; (*Variable hat den Datentyp UDINT*)
	cVAR_TYPE_LREAL : USINT := 10; (*Variable hat den Datentyp REAL*)
	cVAR_TYPE_REAL : USINT := 8; (*Variable hat den Datentyp REAL*)
	cVAR_TYPE_STRING : USINT := 9; (*Variable hat den Datentyp STRING*)
	cVAR_TYPE_DATE_AND_TIME : USINT := 11; (*Variable hat den Datentyp DATE_AND_TIME*)
	
	// config file
	cTAG_TEMPLATE_E : STRING[80] := '</TEMPLATE>'; (*End Tag*)
	cTAG_TEMPLATE_B : STRING[80] := '<TEMPLATE>'; (*Start Tag*)
	cTAG_ROW_E : STRING[80] := '</ROW>'; (*End Tag*)
	cTAG_ROW_B : STRING[80] := '<ROW>'; (*Start Tag*)
	cTAG_RECORD_E : STRING[80] := '</RECORD>'; (*End Tag*)
	cTAG_RECORD_B : STRING[80] := '<RECORD>'; (*Start Tag*)
	cTAG_ITEM_E : STRING[80] := '</ITEM>'; (*End Tag*)
	cTAG_ITEM_B : STRING[80] := '<ITEM>'; (*Start Tag*)
	cTAG_HEADER_E : STRING[80] := '</HEADER>'; (*End Tag*)
	cTAG_HEADER_B : STRING[80] := '<HEADER>'; (*Start Tag*)
	cTAG_FOOTER_E : STRING[80] := '</FOOTER>'; (*End Tag*)
	cTAG_FOOTER_B : STRING[80] := '<FOOTER>'; (*Start Tag*)
	cTAG_CONFIG_E : STRING[80] := '</CONFIG>'; (*End Tag*)
	cTAG_CONFIG_B : STRING[80] := '<CONFIG>'; (*Start Tag*)
	
	// config tags
	cTAG_CFG_LOGFILE_PRAEFIX_E : STRING[80] := '</LOGFILE_PRAEFIX>'; (*End Tag*)
	cTAG_CFG_LOGFILE_PRAEFIX_B : STRING[80] := '<LOGFILE_PRAEFIX>'; (*Start Tag*)
	cTAG_CFG_LOGFILE_EXT_E : STRING[80] := '</LOGFILE_EXT>'; (*End Tag*)
	cTAG_CFG_LOGFILE_EXT_B : STRING[80] := '<LOGFILE_EXT>'; (*Start Tag*)
	cTAG_CFG_QUEUE_LEN_E : STRING[80] := '</QUEUE_LEN>'; (*End Tag*)
	cTAG_CFG_QUEUE_LEN_B : STRING[80] := '<QUEUE_LEN>'; (*Start Tag*)
	cTAG_CFG_LOGTYPE_E : STRING[80] := '</LOG_TYPE>'; (*End Tag*)
	cTAG_CFG_LOGTYPE_B : STRING[80] := '<LOG_TYPE>'; (*Start Tag*)
	cTAG_CFG_MASK_E : STRING[80] := '</LOG_MASK>'; (*End Tag*)
	cTAG_CFG_MASK_B : STRING[80] := '<LOG_MASK>'; (*Start Tag*)
	cTAG_CFG_MAX_LOGFILES_E : STRING[80] := '</MAX_LOGFILES>'; (*End Tag*)
	cTAG_CFG_MAX_LOGFILES_B : STRING[80] := '<MAX_LOGFILES>'; (*Start Tag*)
	cTAG_CFG_T_CHECK_MAX_FILE_NR_E : STRING[80] := '</TIME_CHECK_MAX_FILE_NR>'; (*End Tag*)
	cTAG_CFG_T_CHECK_MAX_FILE_NR_B : STRING[80] := '<TIME_CHECK_MAX_FILE_NR>'; (*Start Tag*)
	cTAG_CFG_MAX_T_TO_WRITE_E : STRING[80] := '</MAX_TIME_TO_WRITE>'; (*End Tag*)
	cTAG_CFG_MAX_T_TO_WRITE_B : STRING[80] := '<MAX_TIME_TO_WRITE>'; (*Start Tag*)
	cTAG_CFG_NEW_FILE_RESTART_E : STRING[80] := '</NEW_FILE_ON_RESTART>'; (*End Tag*)
	cTAG_CFG_NEW_FILE_RESTART_B : STRING[80] := '<NEW_FILE_ON_RESTART>'; (*Start Tag*)
	cTAG_CFG_MAX_ENTR_IN_FILE_E : STRING[80] := '</MAX_ENTRIES_IN_FILE>'; (*End Tag*)
	cTAG_CFG_MAX_ENTR_IN_FILE_B : STRING[80] := '<MAX_ENTRIES_IN_FILE>'; (*Start Tag*)
	cTAG_CFG_MAX_FILE_SIZE_E : STRING[80] := '</MAX_FILE_SIZE>'; (*End Tag*)
	cTAG_CFG_MAX_FILE_SIZE_B : STRING[80] := '<MAX_FILE_SIZE>'; (*Start Tag*)
	cTAG_CFG_LOG_TIMESTAMP_E : STRING[80] := '</LOG_TIMESTAMP>'; (*End Tag*)
	cTAG_CFG_LOG_TIMESTAMP_B : STRING[80] := '<LOG_TIMESTAMP>'; (*Start Tag*)
	cTAG_CFG_LOGFILE_SNETID_E : STRING[80] := '</LOGFILE_SNETID>'; (*End Tag*)
	cTAG_CFG_LOGFILE_SNETID_B : STRING[80] := '<LOGFILE_SNETID>'; (*Start Tag*)
	cTAG_CFG_LOGFILE_PATH_E : STRING[80] := '</LOGFILE_PATH>'; (*End Tag*)
	cTAG_CFG_LOGFILE_PATH_B : STRING[80] := '<LOGFILE_PATH>'; (*Start Tag*)
	cLOG_TIMESTAMP_WIN : STRING[80] := 'LOCAL_TIME'; (*using local time (windows time with time zone)*)
	cLOG_TIMESTAMP_UTC : STRING[80] := 'UTC'; (*using UTC*)
	
	//<ITEM>***</ITEM> predefined items of base log
	cITEM_UNIX_DATE_TIME_STR : STRING[80] := 'DT_UNIX_STR'; (*Item UNIX Datum/Zeit als String*)
	cITEM_UNIX_DATE_TIME : STRING[80] := 'DT_UNIX'; (*Item UNIX Datum/Zeit als Integer*)
	cITEM_TIME_MILLI : STRING[80] := 'TIME_MILLI'; (*Item Millisekunden*)
	cITEM_EXCEL_DATE_TIME : STRING[80] := 'DT_EXCEL'; (*Item date/time in Excel format. Days as real since 1.1.1980*)
	cITEM_DATE_SLASH_TIME_COLON : STRING[80] := 'DATE_SLASH_TIME_COLON'; //english date format 2014/09/23 07:10:24
	cITEM_BL_LOGTYP : STRING[80] := 'BL_LOGTYP'; (*Base Log Item LogTyp*)
	cITEM_BL_CTRL_ID : STRING[80] := 'BL_CTRL_ID'; (*Base Log Item Controller Id*)
	cITEM_BL_STRING1 : STRING[80] := 'BL_STRING1'; (*Base Log Item STRING 1*)
	cITEM_BL_STRING2 : STRING[80] := 'BL_STRING2'; (*Base Log Item STRING 2*)
	cITEM_BL_PAR1 : STRING[80] := 'BL_PAR1'; (*Base Log Item PAR1  *)
	cITEM_BL_PAR2 : STRING[80] := 'BL_PAR2'; (*Base Log Item PAR2*)
	cITEM_BL_PAR3 : STRING[80] := 'BL_PAR3'; (*Base Log Item PAR3*)
	cITEM_BL_PAR4 : STRING[80] := 'BL_PAR4'; (*Base Log Item PAR4*)
	
	// <LOG_TYPE>****</LOG_TYPE>	 predefined values
	cLOGTYP_BL_STR : STRING[80] := 'BL'; (*BaseLog*)
	cLOGTYP_PV_STR : STRING[80] := 'PV'; (*PVLog*)
	cLOGTYP_DATA_STR : STRING[80] := 'DATA'; (*DataLog*)
	cLOGTYP_OPEN_STR : STRING[80] := 'OPEN'; (*Item date/time in Excel format. Days as real since 1.1.1970*)
	
	// Defaults
	cLOGTYP_BL : USINT := 1; (*Baselog*)
	cLOGTYP_PV : USINT := 2; (*PV*)
	cLOGTYP_DATA : USINT := 3; (*Data*)
	cLOGTYP_OPEN : USINT := 4; (*Open --> Maske setzen!*)
	cPVTYPE_UNIX_DATE_TIME_STR : DINT := -3;
	cPVTYPE_UNIX_DATE_TIME : DINT := -1;
	cPVTYPE_DATE_SLASH_TIME_COLON : DINT := -13; //english date format 2014/09/23 07:10:24
	cPVTYPE_TIME_MILLI : DINT := -2;
	cPVTYPE_EXCEL_DATE_TIME : DINT := -4;
	cPVTYPE_BL_LOGTYP : DINT := -5;
	cPVTYPE_BL_CTRL_ID : DINT := -6;
	cPVTYPE_BL_STRING1 : DINT := -7;
	cPVTYPE_BL_STRING2 : DINT := -8;
	cPVTYPE_BL_PAR1 : DINT := -9;
	cPVTYPE_BL_PAR2 : DINT := -10;
	cPVTYPE_BL_PAR3 : DINT := -11;
	cPVTYPE_BL_PAR4 : DINT := -12;
	cTIME_CHECK_MAX_FILE_NR : UDINT := 300; //[s] time period until check number of files in folder
	cMAX_ITEM_CHAR : UINT := BasLog.cMAX_CHAR_TEXT1; (*25 ist das absolute Minimum für DATE_AND_TIME - String Darstellung*)
	cEOL : ARRAY[0..1] OF BYTE := [13,10]; (*End of Line (Line feed, carriage return)*)
	cCMD_FLUSHBUF_NEWFILE : USINT := 2;
	cCMD_FLUSHBUF : USINT := 1;
	cCFG_TIME_WRITE_TO_FILE : UDINT := 60; (*DEFAULT: Mindestens alle 60 Sekunden ins File schreiben*)
	cCFG_QUEUE_LEN : UDINT := 512; (*DEFAULT: Anzahl Elemente der Log Queue*)
	cCFG_LOGFILE_NAME : STRING[80] := 'LogData_'; (*DEFAULT: LogFile Präfix*)
	cCFG_LOGFILE_EXT : STRING[80] := 'txt'; (*DEFAULT: LogFile Extension*)
	cCFG_DEFAULT_MASK : UDINT := 16#FFFFFFFF; // Default mask
	cCFG_MAX_NBR_OF_LOGFILES : UINT := 2; // Defaultmax number of log files
	
	// limits
	cPRE_POST_TEXTLEN : UINT := 256; // max text len for pre and post text of a value
	cMAX_RECORDS_IN_FILE_BUF : UINT := 4; (*factor for calculation of file buffer*)
	cMAX_NBR_OF_FILECLIENTS : UINT := 10; (*Max number of file clients*)
	cFILENAME_LENGTH : UINT := 260; // config file name len
	cPATH_LENGTH : UINT := 260; // folderpath string len
	
	// error number	
	cERR_NBR_OF_FC_EXEEDED : UINT := 50400; (*Max number of file clients reached*)
	cERR_FILENAME_MISSING : UINT := 50401; (*Filename missing*)
	cERR_PATH_MISSING : UINT := 50402; (*Path definition missing*)
	cERR_CONFIG_TAG : UINT := 50403; (*Error in <CONFIG></CONFIG> tag*)
	cERR_TEMPLATE_TAG : UINT := 50404; (*Error in <TEMPLATE></TEMPLATE> tag*)
	cERR_INVALID_LOGTYP : UINT := 50405; (*Unknown or missing log type -> template/config - file*)
	cERR_HEADER_TAG : UINT := 50406; (*Error in <HEADER></HEADER> tag*)
	cERR_RECORD_TAG : UINT := 50407; (*Error in <RECORD></RECORD> tag*)
	cERR_ROW_TAG : UINT := 50408; (*Error in <ROW></ROW> tag*)
	cERR_ITEM_TAG : UINT := 50409; (*Error in <ITEM></ITEM> tag*)
	cERR_FOOTER_TAG : UINT := 50410; (*Error in <FOOTER></FOOTER> tag*)
	cERR_HANDLE : UINT := 50411; (*no handle reached*)
	cERR_INVALID_DEVICE : UINT := 50412; (*File destination not correct*)
	cERR_ALLOC_BUFFER_FILE_CONFIG : UINT := 50413; (*No memory available for config read out*)
	cERR_ALLOC_MEMORY : UINT := 50414; (*No memory available*)
	cERR_NO_BASELOG : UINT := 50415; (*BaseLog pointer invalid*)
	cERR_NO_FLCIDX : UINT := 50416; (*INIT not possibel no valid act client nr index reference / pointer invalid*)
END_VAR

// POUs/Utility/Queue/Queue
VAR_GLOBAL CONSTANT
	// internal
	cSECURE_CODE: UDINT := 1431655765; // alternating bit muster 0x55555555 -> for validation of queues
	
	// limits
	cMAX_NAME_LENGTH : UINT := 80; // maximal string length of queue name
	cMAX_NR_OF_TASKS: USINT := 6; // for the moment enough

	// error number
	cERR_QUEUE_FULL : UINT := 1; 
	cERR_QUEUE_EMPTY : UINT := 2; 
	cERR_QUEUE_NAME : UINT := 50000; // not valid or empty queue name
	cERR_NR_OF_ELEMENTS : UINT := 50001; // number of elements =0 
	cERR_SIZE_OF_ELEMENTS: UINT := 50002; // element size =0
	cERR_MEM_ALLOC  : UINT := 50003; // error allocate memory
	cERR_QUEUE_DOES_NOT_EXIST : UINT := 50004; // queue does not exist
	cERR_Q_INFO_DOES_NOT_EXIST : UINT := 50005; // queue info does not exist
	cERR_DATA_INVALID : UINT := 50006; // pointer to data not valid
	cERR_HANDLE_INVALID : UINT := 50007; // handle not ok
	cERR_TC_INVALID : UINT := 50008; // task class index not ok
	cERR_CLEAR : UINT := 50009; // clear of queue not ok
END_VAR

// Version/Global_Version
// This function has been automatically generated from the project information.
VAR_GLOBAL CONSTANT
	{attribute 'const_non_replaced'}
	stLibVersion_Base_PLC : ST_LibVersion := (iMajor := 0, iMinor := 3, iBuild := 5, iRevision := 10, sVersion := '0.3.5.10');
END_VAR

// POUs/Alarm/FB_Alm_Man
FUNCTION_BLOCK FB_Alm_Man
VAR_INPUT
	;
END_VAR
VAR_IN_OUT
	bolCtrlRst: BOOL; // reset all controller
END_VAR

VAR CONSTANT
	/// config alarm handler number of elements of queue
	c_uinMaxAlmElements: UINT := 99;
	/// 0: with history on PLC, auto clr alarms from array if alarm state clear is set
	c_uinModeAlarm: UINT := 1;
	/// machine number 1, at the moment every time set to 1
	c_udiMachineNr: UDINT := 1;
	/// commands from the UI
	cCMD_RESET_ALL: INT := 2;
	/// reset state=RST, reset state CLR
	cCMD_RESET_RST: INT := 4;
	/// reset state CLR -> c_uinModeAlarm = 1, automatic reset will be done on PLC
	cCMD_RESET_CLR: INT := 6;
END_VAR
VAR
	///------------------------------------------------------------
	/// UI interface
	/// alarmarray PLC -> UI
	aAlm: ARRAY[0..c_uinMaxAlmElements] OF T_AlmElement;
	/// command interface for UI -> PLC
	intAlmCmd: INT;
	///------------------------------------------------------------
	fbTimeStamp: FB_TimeStamp; // only one central time for time stamps

	jj: UINT;
	EmptyAlmElement: T_AlmElement;
	intState: INT;
	intTestCtrl: INT := 12;
	intTestState: INT;
	udiTestAlarmNr: UDINT;
	dinTestInfo: DINT;
	aCtrlAlm: ARRAY[1..6] OF T_Ctrl_Alm;
	eActiveAlmClass: E_AlmClass;

	aCntActiveAlmPerClass: ARRAY[0..(E_AlmClass.Max_E_AlmClass-1)] OF UINT; // count off all active alarms per class, idx=0 all active alarms
END_VAR

(*__________________________________________________________________________________________________
¦	
¦	Vistaprint Schweiz GmbH
¦	CH - 8401 Winterthur
¦
¦	www.vistaprint.ch - info@vistaprint.ch
¦___________________________________________________________________________________________________

Function desription:
The alarm manager sets and clears alarms from the internal array. In the internal array all active 
alarms of a machine are listed. The list has no order. A new entry will be inserted at the next 
free place.

For the easy usage for UI the function block is to be define as global. And then the cmd for reset should be 
set when the button is pressed -> intAlmCmd = cCMD_RESET_ALL
All active alarms are shown in the aAlm array.

History:
Version		Date			Author		Comment
---------------------------------------------------------------------------------------------------
0.00.1		29.04.2013		AVME/KVO	Start history
0.00.2		06.01.2014		AVME/PRE	Implement the counted active messages array
0.00.3		17.02.2014		AVME/KVO	New Property IsInitDone 
										feedback at least one valid time stamp read out 
										-> check at startup before cyclic call of FB's to avoid alarms without valid timestamp
0.00.4		16.05.2014		AVME/DSC	-> Inserted new "setAlarm" Method from Patrik C. (code review)									
										-> BugFix, build sum of all active alarms
0.00.5		07.07.2014		AVME/KVO	-> BugFix Method setAlarm , clr and reset -> also possibel if one entry is zero possibel
0.00.6		07.10.2014		AVME/KVO	-> BugFix alarm reset first statemachine and then the messages	
0.00.7		27.10.2014		AVME/KVO	-> delete GETSYSTEMTIME use FB_TimeStamp
										-> New time properties for easy access of every controller if needed
___________________________________________________________________________________________________*)

// call time stamp asynchronous synchronisation
fbTimeStamp.In_strNetId := ''; // use system time of log target system
fbTimeStamp.In_t_CycleTimeRefreshTimeZone := T#0S; // cyclic check time zone settings - not needed using LocalTime_FileTime_BaseWin for log system and local time
fbTimeStamp();

// interface for UI access
CASE intState OF
		
	0: // reset cmd
		intAlmCmd := cCMD_DONE; // Ready for new cmd
		intState := intState + 1;
		
	1: // wait for cmd
		IF (intAlmCmd=cCMD_RESET_ALL) OR (intAlmCmd=cCMD_RESET_CLR) OR  (intAlmCmd=cCMD_RESET_RST) THEN
			intState := intState + 1;
		END_IF
		
	2: // firt reset state machines -> leave Error state
		bolCtrlRst := TRUE;
		intState := intState + 1;
		
	3: // reset alarms / messages
		// reset state=RST, reset state CLR
		THIS^.clearAlarm(((intAlmCmd=cCMD_RESET_ALL) OR (intAlmCmd=cCMD_RESET_RST)), TRUE);
		intState := intState + 1;
		
	4: 
		intState := 0; // done
END_CASE

// build sum of all active alarms
aCntActiveAlmPerClass[0] := 0;
FOR jj:= 1 TO INT_TO_UINT(E_AlmClass.Max_E_AlmClass-1) BY 1 DO
	aCntActiveAlmPerClass[0] := aCntActiveAlmPerClass[0] + aCntActiveAlmPerClass[jj];
END_FOR

//**********************************************************************************************
// Test manual set/reset/clear alarm
//**********************************************************************************************
CASE intTestState OF
	
	0: // wait
		
	1: //CLR
		THIS^.setAlarm(intTestCtrl,udiTestAlarmNr,dinTestInfo,ADR(aCtrlAlm),E_AlmState.CLR,eActiveAlmClass);
		intTestState := 0;
		
	2: // RST
		THIS^.setAlarm(intTestCtrl,udiTestAlarmNr,dinTestInfo,ADR(aCtrlAlm),E_AlmState.RST,eActiveAlmClass);
		intTestState := 0;
		
	3: // SET
		THIS^.setAlarm(intTestCtrl,udiTestAlarmNr,dinTestInfo,ADR(aCtrlAlm),E_AlmState.SET,eActiveAlmClass);
		intTestState := 0;

END_CASE

PROPERTY PUBLIC aCntPerClass : ARRAY[0..(E_AlmClass.Max_E_AlmClass-1)] OF UINT
GET
aCntPerClass := aCntActiveAlmPerClass;
END_GET
END_PROPERTY

METHOD clearAlarm : BOOL
VAR_INPUT
	///-> clear all entries with state RST
	bolClear_RST: BOOL;
	///-> clear all entries with state CLR
	bolClear_CLR: BOOL;
END_VAR
VAR
	ii: UINT;
END_VAR
FOR ii:= 0 TO INT_TO_UINT(E_AlmClass.Max_E_AlmClass-1) BY 1 DO
	aCntActiveAlmPerClass[ii] := 0; // reset alarm counter
END_FOR

FOR ii:= 0 TO c_uinMaxAlmElements BY 1 DO
	
	IF (aAlm[ii].udiNr>0) THEN 
		
		IF (((aAlm[ii].intState=E_AlmState.RST) AND (bolClear_RST)) OR
			((aAlm[ii].intState=E_AlmState.CLR) AND (bolClear_CLR)))THEN
			
			aAlm[ii] := EmptyAlmElement; // clear entry
		ELSE
			//count alarms per class
			aCntActiveAlmPerClass[aAlm[ii].eClass] := aCntActiveAlmPerClass[aAlm[ii].eClass] + 1; 
		END_IF
		
	END_IF
END_FOR
END_METHOD

PROPERTY IsInitDone : BOOL
GET
// feedback at least one valid time stamp read out 
//-> check at startup before cyclic call of FB's to avoid alarms without valid timestamp
IsInitDone := fbTimeStamp.Out_bolInitOk;
END_GET
END_PROPERTY

PROPERTY PUBLIC LocalTime_FileTime_BaseWin : T_FileTime
GET
VAR
	fbToLocal : FB_FileTimeToTzSpecificLocalTime;
END_VAR
LocalTime_FileTime_BaseWin := fbTimeStamp.LocalTime_FileTime_BaseWin;
END_GET
END_PROPERTY

PROPERTY PUBLIC LocalTime_TimeStruct_BaseWin : TIMESTRUCT
GET
LocalTime_TimeStruct_BaseWin :=fbTimeStamp.LocalTime_TimeStruct_BaseWin;
END_GET
END_PROPERTY

METHOD setAlarm : E_AlmClass
VAR_INPUT
	///from controller 
	intCtrlId: INT;
	///local alarm number
	udiAlarmNr: UDINT;
	///additional information - string???
	dinInfo: DINT;
	///corresponding alarm class
	p_Ctrl_Alm: POINTER TO T_Ctrl_Alm;
	///clear, resetable
	intState: E_AlmState;
END_VAR
VAR_IN_OUT
	eMe_ActivAlmClass: E_AlmClass;
END_VAR
VAR
	InAlmElement: T_AlmElement;
	ii: UINT;
	uinFirstEmptyIdx : UINT;
	e_LocAlmClass: E_AlmClass;
END_VAR
// chack if pointer valid
IF (p_Ctrl_Alm <> Tc3_MemMan.NULL) AND (udiAlarmNr>0) THEN 
	e_LocAlmClass := p_Ctrl_Alm[udiAlarmNr-1].eAlmClass;
ELSE
	// novalid pointer reached!!
   	e_LocAlmClass := E_AlmClass.EOFF; 
END_IF
 
// Copy alarm input data to local alm struct
InAlmElement.udiMachineNr := c_udiMachineNr;
InAlmElement.intCtrlId := intCtrlId;
InAlmElement.udiAlarmNr := udiAlarmNr;
InAlmElement.udiNr := 100000*InAlmElement.udiMachineNr + INT_TO_UDINT(100*InAlmElement.intCtrlId) + InAlmElement.udiAlarmNr;
InAlmElement.dinInfo := dinInfo;
InAlmElement.eClass := e_LocAlmClass;
InAlmElement.intState := intState;
// YYYY-MM-DD-hh:mm:ss.xxx
InAlmElement.strDTEntry := TC2_UTILITIES.SYSTEMTIME_TO_STRING(fbTimeStamp.LocalTime_TimeStruct_BaseWin);
InAlmElement.strText := p_Ctrl_Alm[udiAlarmNr-1].strText;

ii := 0;
uinFirstEmptyIdx := c_uinMaxAlmElements + 1;
//KVO 7.7.2014 AND (aAlm[ii].udiNr <> 0) removed from while because there could be entries above a cleared alarm!
WHILE (ii <= c_uinMaxAlmElements)  AND (InAlmElement.udiNr <> aAlm[ii].udiNr) DO
	IF (aAlm[ii].udiNr = 0) AND (uinFirstEmptyIdx>c_uinMaxAlmElements) THEN // entry first empty index
		uinFirstEmptyIdx := ii;
	END_IF
	ii := ii + 1;              
END_WHILE

// set ii to first empty place (new entry) in array if entry not allready exists in array
IF (uinFirstEmptyIdx<= c_uinMaxAlmElements) AND (InAlmElement.udiNr <> aAlm[ii].udiNr) THEN
	ii := uinFirstEmptyIdx;
END_IF

IF (ii <= c_uinMaxAlmElements) THEN
	
	// Alarm already exist
	IF (aAlm[ii].udiNr = InAlmElement.udiNr) THEN
		CASE InAlmElement.intState OF
			E_AlmState.SET, E_AlmState.RST:
				// refresh state, alarm additional info
				aAlm[ii].dinInfo := InAlmElement.dinInfo;
				aAlm[ii].intState := InAlmElement.intState;
			E_AlmState.CLR:
				IF (aCntActiveAlmPerClass[aAlm[ii].eClass]>0) THEN
					aCntActiveAlmPerClass[aAlm[ii].eClass] := aCntActiveAlmPerClass[aAlm[ii].eClass] - 1; 
				END_IF
				
				IF (c_uinModeAlarm=1) THEN // no history on PLC
					aAlm[ii] := EmptyAlmElement; // clear entry
				ELSE
					aAlm[ii].intState := E_AlmState.CLR; // set clear state -> entry in plc history if needed
				END_IF
		END_CASE          
	END_IF
	
	// New Alarm entry
	IF (aAlm[ii].udiNr = 0) THEN
		CASE InAlmElement.intState OF
			E_AlmState.SET, E_AlmState.RST:
				aAlm[ii] := InAlmElement;
				//count alarms per class
				aCntActiveAlmPerClass[aAlm[ii].eClass] := aCntActiveAlmPerClass[aAlm[ii].eClass] + 1; 
	
				IF (InAlmElement.eClass>eMe_ActivAlmClass) THEN 
					eMe_ActivAlmClass := InAlmElement.eClass;
				END_IF
		END_CASE
	END_IF
	
END_IF
END_METHOD

PROPERTY PUBLIC UTC_FileTime : T_FileTime
GET
VAR
	fbGETSYSTEMTIME : GETSYSTEMTIME;
END_VAR
UTC_FileTime := fbTimeStamp.UTC_FileTime;
END_GET
END_PROPERTY

PROPERTY PUBLIC UTC_TimeStruct : TIMESTRUCT
GET
UTC_TimeStruct := fbTimeStamp.UTC_TimeStruct;
END_GET
END_PROPERTY

END_FUNCTION_BLOCK

// POUs/Utility/FB_TimeStamp
FUNCTION_BLOCK PUBLIC FB_TimeStamp
VAR_INPUT
		In_t_CycleTimeRefreshTimeZone : TIME;
		In_strNetId : T_AmsNetID;
END_VAR
VAR_OUTPUT
	Out_bolInitOk : BOOL; // init ok  (i.e. it was synchronised with the local Windows time at least once).
END_VAR
VAR
	tzID    : E_TimeZoneID; // Additional daylight-saving/standard time information (not always existent)
    tzInfo  : ST_TimeZoneInformation; //In case of success this structure variable supplies the current time zone information of the operating system.
	fbTONRefreshTimeZone : TON;
	bolSuccessfullyDone : BOOL;
	bolStartGetTimeZone : BOOL;
	udiError : UDINT;
	fbGetTimeZoneInformation: FB_GetTimeZoneInformation;
	fbToLocal : FB_FileTimeToTzSpecificLocalTime;
	fbLocalTime : FB_LocalSystemTime := ( bEnable := TRUE, dwCycle := 1 ,dwOpt := 1);
	fbLocalTime_RTC : RTC_EX2;
    //dwOpt: Bit 0: If this is set, the Windows system time is additionally synchronised cyclically with the hardware clock (RTC) (corresponds to the function NT_SetTimeToRTCTime). Default: Activated.
    //This option is irrelevant for a Windows CE system.

	bolStartUp : BOOL := TRUE;
	bolInitTimeZoneOk  : BOOL := FALSE;
END_VAR

(*__________________________________________________________________________________________________
¦	
¦	Vistaprint Schweiz GmbH
¦	CH - 8401 Winterthur
¦
¦	www.vistaprint.ch - info@vistaprint.ch
¦___________________________________________________________________________________________________

Function desription:
Idea of this FUB is a central solution to get time stamps on PLC synchronized with windows time. 

Automatic synchronisation of the RTC time using the function block "NT_SetTimeToRTCTime" 
an be used to synchronise the local Windows system time (displayed in the task bar) with the real-time clock of the PC (RTC time in the BIOS). 
At System startup this system synchronisation will be done.

Properties only read:
Cyclic FB call is needed for automatic time zone synchronisation, local time calculation, changes, adjustments  on windows time not detected!
-> LocalTime_FileTime_BaseUTC : Before get call UTC_Refresh! data typ FileTime in local time calculated based on time zone and on UTC FileTime 
-> LocalTime_TimeStruct_BaseUTC : Before get call UTC_Refresh! data typ TimeStruct in local time calculated based on time zone and on UTC FileTime 

Not use for exact measurements because of automatic asynchron windows synchronisation(the local Windows system time is displayed in the task bar)!
Cyclic FB call is needed for automatic windows synchronisation of win time!
-> LocalTime_FileTime_BaseWin : automatic refresh on get, data typ FileTime in windows time shown in taskbar. 
-> LocalTime_TimeStruct_BaseWin : automatic refresh on get, data typ TimeStruct in windows time shown in taskbar

-> UTC_FileTime : automatic refresh on get, data typ FileTime in UTC 
-> UTC_TimeStruct :  automatic refresh on get, data typ TimeStruct in UTC 

Methods:
-> TimeZone_Refresh : Refreh time zone information -> for  explicit time calculation  UTC<->Win

FB Cyclic: 
	- automatic FB_LocalSystemTime asynchron windows time synchronisation for LocalTime_FileTime_BaseWin/LocalTime_TimeStruct_BaseWin needed
	- automatic cyclic TimeZone_Refresh based on In_t_CycleTimeRefreshTimeZone parameter if =0 -> disabled

History:
Version		Date			Author		Comment
---------------------------------------------------------------------------------------------------
0.00.1		10.10.2014		AVME/KVO	Start history

___________________________________________________________________________________________________*)

// refresh time Zone
IF ((In_t_CycleTimeRefreshTimeZone<>T#0S)OR (bolStartUp=TRUE)) THEN
	// cylic call of FUB will automatic cyclic refresh the Time Zone informations
	IF (fbTONRefreshTimeZone.IN = FALSE) THEN
		fbTONRefreshTimeZone();
		fbTONRefreshTimeZone.IN := TRUE;
		fbTONRefreshTimeZone.PT := In_t_CycleTimeRefreshTimeZone;
		bolSuccessfullyDone := FALSE;
		udiError := 0; // reset last alarm
	END_IF
	
	fbTONRefreshTimeZone();
	
	// Zeit abgelaufen
	IF (fbTONRefreshTimeZone.Q) OR (bolStartUp=TRUE) THEN
		IF ((bolSuccessfullyDone=FALSE) AND (udiError=0)) THEN
			udiError := TimeZone_Refresh(In_strNetId :=In_strNetId,Out_bolSuccessfullyDone=> bolSuccessfullyDone);
		ELSE
			bolStartUp := FALSE; // FirstCycle DirectionParameterOverflow call -> refresh!!
			bolInitTimeZoneOk := TRUE;
			fbTONRefreshTimeZone.IN := FALSE; // start next cycle
		END_IF
	END_IF
END_IF

//The FB_LocalSystemTime function block must be called cyclically (e.g. every second or during each PLC cycle). 
//This is necessary to enable the time between synchronisations to be calculated.
(*The local Windows system time is read with the aid of acyclic services (ADS function blocks). 
Due to the system characteristics the runtime of the ADS commands cannot be specified/estimated. 
Differences in command runtimes may lead to time jitter at the systemTime output, depending on the operating system, 
the synchronisation interval and the PLC cycle time. For this reason the time supplied by the 
block is only suitable to a limited extent for measuring tasks requiring higher precision, 
although it tends to be adequate for building automation applications, for example.*)

(*This function block internally combines the functions of the following function blocks: RTC_EX2, NT_GetTime, FB_GetTimeZoneInformation and NT_SetTimeToRTCTime. 
The RTC_EX2 block can be used for generating time stamps for log outputs, for example. 
However, this block has the disadvantage that its time is not synchronised with the local Windows system time and has to be resynchronised 
cyclically via the NT_GetTime function block (see RTC block examples in the documentation). Cyclic synchronisation of the internal time (systemTime output) 
is already implemented in the function block. 
The cycle time can be configured via the dwCycle input. The function block also provides time zone information (daylight-saving/standard time).*)
fbLocalTime.sNetID := In_strNetId;
fbLocalTime(); // for local time it seems to be ok for logging (not measuring), for exact measuring it's simpler to just use the utc time!!!!

// synchronize RTC for fast access
IF (fbLocalTime.bValid = TRUE) THEN
	fbLocalTime_RTC.EN := FALSE;
	fbLocalTime_RTC();
	fbLocalTime_RTC.EN := TRUE;
	fbLocalTime_RTC.PDT := fbLocalTime.systemTime;
	fbLocalTime_RTC.PMICRO := 0;
	fbLocalTime_RTC();
END_IF

Out_bolInitOk := ((fbLocalTime.bValid=TRUE) AND (bolInitTimeZoneOk=TRUE) AND (fbLocalTime_RTC.Q=TRUE));

PROPERTY PUBLIC LocalTime_FileTime_BaseUTC : T_FileTime
GET
// use before/last refreshed UTC as base and calculates based on the UTC and the time zone -> the local time
fbToLocal.in := UTC_FileTime;
fbToLocal.tzInfo := tzInfo;
fbToLocal(); // tests -> is exact but if a user change the windows time no change on this time stamp
LocalTime_FileTime_BaseUTC :=fbToLocal.out;
END_GET
END_PROPERTY

PROPERTY PUBLIC LocalTime_FileTime_BaseWin : T_FileTime
GET
VAR
	fbToLocal : FB_FileTimeToTzSpecificLocalTime;
END_VAR
LocalTime_FileTime_BaseWin := SYSTEMTIME_TO_FILETIME( LocalTime_TimeStruct_BaseWin );
END_GET
END_PROPERTY

PROPERTY PUBLIC LocalTime_TimeStruct_BaseUTC : TIMESTRUCT
GET
LocalTime_TimeStruct_BaseUTC := FILETIME_TO_SYSTEMTIME( LocalTime_FileTime_BaseUTC );
END_GET
END_PROPERTY

PROPERTY PUBLIC LocalTime_TimeStruct_BaseWin : TIMESTRUCT
GET
// for local time it seems to be ok for logging (not measuring), for exact measuring it's simpler to just use the utc time!!!!
//fbLocalTime(); make some trouble if called in fast tk -> use seperate RTC!!!!
fbLocalTime_RTC();
LocalTime_TimeStruct_BaseWin := fbLocalTime_RTC.CDT; //fbLocalTime.systemTime;
END_GET
END_PROPERTY

METHOD PUBLIC TimeZone_Refresh : UDINT
VAR_INPUT
	In_strNetId : T_AmsNetID;
END_VAR
VAR_OUTPUT
	Out_bolSuccessfullyDone : BOOL;
END_VAR
// reads out the windows time zone
IF (bolStartGetTimeZone = FALSE) THEN
	fbGetTimeZoneInformation.bExecute := FALSE;
	fbGetTimeZoneInformation();
	fbGetTimeZoneInformation.sNetID  := In_strNetId;
	fbGetTimeZoneInformation.bExecute := TRUE;
	fbGetTimeZoneInformation();
	bolStartGetTimeZone := TRUE; 
ELSE
	fbGetTimeZoneInformation();
	IF (fbGetTimeZoneInformation.bBusy=FALSE) THEN
		IF (fbGetTimeZoneInformation.bError=FALSE) THEN
			tzID := fbGetTimeZoneInformation.tzID;
        	tzInfo := fbGetTimeZoneInformation.tzInfo;
			Out_bolSuccessfullyDone := TRUE;
		ELSE
			TimeZone_Refresh := fbGetTimeZoneInformation.nErrID;
		END_IF
		bolStartGetTimeZone := FALSE;
	END_IF
END_IF
END_METHOD

PROPERTY PUBLIC UTC_FileTime : T_FileTime
GET
VAR
	fbGETSYSTEMTIME : GETSYSTEMTIME;
END_VAR
// read out actual TIME in UTC (NT_GETTIME needs to much cycles!!!!!)
fbGETSYSTEMTIME(timeLoDW=>UTC_FileTime.dwLowDateTime, timeHiDW=>UTC_FileTime.dwHighDateTime); // UTC available in one cycle
END_GET
END_PROPERTY

PROPERTY PUBLIC UTC_TimeStruct : TIMESTRUCT
GET
UTC_TimeStruct := FILETIME_TO_SYSTEMTIME(UTC_FileTime);
END_GET
END_PROPERTY

END_FUNCTION_BLOCK

// POUs/BaseCtrl/FB_CtrlBase
{attribute 'reflection'}
FUNCTION_BLOCK FB_CtrlBase IMPLEMENTS I_CtrlBase
VAR
	// common interface struct for public access
	CIf						: T_Ctrl_CIf;

	{attribute 'noinit'}
	{attribute 'instance-path'}
	strMyInstancePath: STRING;

	// pointer to global alarm handler function block 
	pfbAlarmCtrl			: POINTER TO FB_Alm_Man;
	
	// basic local controller class struct
	me						: T_Ctrl_Class;
	fbSimulationTimer		: TON;
END_VAR

(*__________________________________________________________________________________________________
¦	
¦	Vistaprint Schweiz GmbH
¦	CH - 8401 Winterthur
¦
¦	www.vistaprint.ch - info@vistaprint.ch
¦___________________________________________________________________________________________________

Function desription:
Basic controller implementation. This Controller should be the base father controller for all in the
feature implemented ctontroller classes.


History:
Version		Date			Author		Comment
---------------------------------------------------------------------------------------------------
0.00.1		25.04.2013		AVME/KVO	Start history
0.00.2		06.01.2014		AVME/PRE	Alarmclasses EOFF, OFF and STOP are send to parent and childs
0.00.3		08.01.2014		AVME/KVO	CheckParentAlmClass OFF and STOP added -> reaction of Controller
0.00.4		04.02.2014		AVME/KVO	New CheckAllChildState also true feedback if check state of 
										child OFF or EOFF and child in ERROR
0.00.5		17.02.2014		AVME/KVO	Bug fix Always Single-answer and startup with wait on PON before change 
										state to EOFFBusy and so on
										Bug fix in CheckParentAlmClass not reset command PON
0.00.6		26.02.2014		AVME/DSC	State single answer. Reset pending alarm class to NONE.
0.00.5		27.10.2014		AVME/KVO	CtrlInit() call set bolInitDone in CtrlInit , allow only one time call CtrlInit, 
										cyclic methode calls only allowed if alarm pointer defined
___________________________________________________________________________________________________*)


IF (me.bolActivate) THEN // cyclic call enabled
	IF (CIf.Info.bolInitDone=FALSE) THEN // first cycle -> only init call if not done before!
		CtrlInit();
	// before go to cyclic the init has to be finished and a valid alarm pointer has to be set
	ELSIF (pfbAlarmCtrl<>0) THEN
		CycleStartDuty();
		Always();
		StateMachine();
		CycleEndDuty();
	END_IF
END_IF;

METHOD PROTECTED AddChild : POINTER TO T_Ctrl_CIf;
VAR_INPUT
	p_fbChild			: I_CtrlBase;
END_VAR
AddChild := 0;

IF CIf.Info.uinChildNbr <= Base_Const.cMaxNrOfChilds THEN
	CIf.Info.p_afbChild[CIf.Info.uinChildNbr] := p_fbChild.CtrlFB;
	CIf.Info.p_aCIf[CIf.Info.uinChildNbr] := CIf.Info.p_afbChild[CIf.Info.uinChildNbr]^.CtrlCIf;
	CIf.Info.p_aCIf[CIf.Info.uinChildNbr]^.Info.intParentCtrlId := CIf.Info.intCtrlId;
	CIf.Info.uinChildNbr := CIf.Info.uinChildNbr + 1;
	AddChild := p_fbChild.CtrlCIf;
END_IF
END_METHOD

PROPERTY PUBLIC AlarmCtrl : POINTER TO FB_Alm_Man
SET
pfbAlarmCtrl := AlarmCtrl;
END_SET
END_PROPERTY

METHOD PROTECTED Always : BOOL
// ----------------------------------------------------------------------------------
// cyclic actions outside of statemachine
IF (me.StateMachine.intState<>cSTA_SINGLE_ANSWER) THEN
	
	// always error supervision
	// ---------------------------------------------------------------------------------
	;
	
END_IF

// ----------------------------------------------------------------------------------
// Conditions Always
IF (me.bolChangeBackToAUTO=TRUE) THEN // switch mode to automatic switch off controller
	me.StateMachine.intStateNext := cSTA_OFFBusy;
	me.bolChangeBackToAUTO := FALSE;
END_IF

IF (CIf.SwCfg.bolExist=FALSE) THEN // hardware of controller does not exist
	me.StateMachine.intStateNext := cSTA_SINGLE_ANSWER;
ELSE
	IF (((me.StateMachine.intState=cSTA_INITIALIZED) OR (me.intCmd=cCMD_PON)) 
		AND (me.StateMachine.intState<>cSTA_PONBusy) AND (me.StateMachine.intState<>cSTA_PON)
		AND (me.StateMachine.intState<>cSTA_ERROR) AND (me.StateMachine.intState<>cSTA_ERRORQuit) 
		AND (me.StateMachine.intState<>cSTA_EOFF) AND (me.StateMachine.intState<>cSTA_EOFFBusy)) THEN // switch after startup to PONBusy
		me.StateMachine.intStateNext := cSTA_PONBusy;
		
	ELSIF ((((NOT me.AlarmConfig.bolEOffAlarmTransitionDisable) AND (me.Alarm.eActivAlmClass=E_AlmClass.EOFF)) OR ((NOT me.AlarmConfig.bolEOffCmdTransitionDisable) AND (me.intCmd=cCMD_EOFF))) 
		AND (me.StateMachine.intState<>cSTA_ERROR) AND (me.StateMachine.intState<>cSTA_ERRORQuit) 
		AND (me.StateMachine.intState<>cSTA_EOFF) AND (me.StateMachine.intState<>cSTA_EOFFBusy)
		AND (me.StateMachine.intState>cSTA_PON)) THEN
		me.StateMachine.intStateNext := cSTA_EOFFBusy;
		
		IF ((NOT me.AlarmConfig.bolEOffAlarmTransitionDisable) AND (me.Alarm.eActivAlmClass=E_AlmClass.EOFF)) THEN
			me.StateMachine.intState := cSTA_DONE;
		END_IF
	
	ELSIF ((((NOT me.AlarmConfig.bolOffAlarmTransitionDisable) AND (me.Alarm.eActivAlmClass=E_AlmClass.OFF)) OR ((NOT me.AlarmConfig.bolOffCmdTransitionDisable) AND (me.intCmd=cCMD_OFF)))
		AND (me.StateMachine.intState<>cSTA_ERROR) AND (me.StateMachine.intState<>cSTA_ERRORQuit)
		AND (me.StateMachine.intState<>cSTA_EOFF) AND (me.StateMachine.intState<>cSTA_EOFFBusy)
		AND (me.StateMachine.intState<>cSTA_OFF) AND (me.StateMachine.intState<>cSTA_OFFBusy)
		AND (me.StateMachine.intState>cSTA_PON)) THEN
		me.StateMachine.intStateNext := cSTA_OFFBusy;
		
		IF ((NOT me.AlarmConfig.bolEOffAlarmTransitionDisable) AND (me.Alarm.eActivAlmClass=E_AlmClass.OFF)) THEN
			me.StateMachine.intState := cSTA_DONE;
		END_IF
		
	ELSE
		FurtherReactions();
	END_IF

	IF CIf.SwCfg.bolAllSimulation AND NOT me.bolSimulateAllExecuted THEN
		SetAllSimulation();
	END_IF
	
	IF NOT CIf.SwCfg.bolAllSimulation AND me.bolSimulateAllExecuted THEN
		ClearAllSimulation();
	END_IF

END_IF
END_METHOD

PROPERTY PUBLIC BaseLog : POINTER TO FB_BasLog
SET
me.stStateLogger.pfbBaseLog := BaseLog;
me.stStateLogger.pHandle:=TC3_MEMMAN.NULL; // reset handle
END_SET
END_PROPERTY

METHOD PROTECTED CheckAllChildAlmClass : BOOL
VAR_INPUT
	In_intCheckAlmClass : INT;
END_VAR
VAR
	uinIdx: UINT;
END_VAR
// check if at least one child has actual this alarm class active
CheckAllChildAlmClass := FALSE;

IF (CIf.Info.uinChildNbr > 0) THEN
	FOR uinIdx := 0 TO CIf.Info.uinChildNbr - 1 DO
		CheckAllChildAlmClass := (CIf.Info.p_aCIf[uinIdx]^.Job.eMe_ActivAlmClass = In_intCheckAlmClass);
		IF (CheckAllChildAlmClass=TRUE) THEN // at least one child has actual this alarm class active
			EXIT;
		END_IF
	END_FOR
END_IF
END_METHOD

METHOD PROTECTED CheckAllChildState : BOOL;
VAR_INPUT
	In_intCheckState : INT;
END_VAR
VAR
	uinIdx: UINT;
END_VAR
// check if all child controller have reached the final In_intCheckState
CheckAllChildState := TRUE;
IF (CIf.Info.uinChildNbr > 0) THEN
	FOR uinIdx := 0 TO CIf.Info.uinChildNbr - 1 DO
		IF ((In_intCheckState<>cSTA_EOFF) AND (In_intCheckState<>cSTA_OFF)) THEN
			CheckAllChildState := CheckAllChildState AND (CIf.Info.p_aCIf[uinIdx]^.Job.intState = In_intCheckState);
		ELSE
			// if controlled state is OFF or EOFF and child is in ERROR -> answer state reached
			CheckAllChildState := (CheckAllChildState AND ((CIf.Info.p_aCIf[uinIdx]^.Job.intState = In_intCheckState) OR (CIf.Info.p_aCIf[uinIdx]^.Job.intState = cSTA_ERROR)));
		END_IF
		IF (CheckAllChildState=FALSE) THEN	// at least one child has not whished state reached
			EXIT ;
		END_IF 
	END_FOR
END_IF
END_METHOD

METHOD CheckChildAlmClass : BOOL
VAR_INPUT
;
END_VAR
VAR
;
END_VAR
//------------------------------------------------------------------------------------------------------
// check child alarm classes
// set me alarm class active if at least one child has an EOFF
IF CheckAllChildAlmClass(E_AlmClass.EOFF) THEN
	CIf.Job.eMe_ActivAlmClass := E_AlmClass.EOFF;
	me.Alarm.bolfp := TRUE;
ELSIF CheckAllChildAlmClass(E_AlmClass.OFF) THEN
	CIf.Job.eMe_ActivAlmClass := E_AlmClass.OFF;
	me.Alarm.bolfp := TRUE;
ELSIF CheckAllChildAlmClass(E_AlmClass.STOP) THEN
	CIf.Job.eMe_ActivAlmClass := E_AlmClass.STOP;
	me.Alarm.bolfp := TRUE;	
ELSE
	IF (me.Alarm.bolfp) THEN
		CIf.Job.eMe_ActivAlmClass := E_AlmClass.NONE; // no reset necessary
		me.Alarm.bolfp := FALSE;
	END_IF
END_IF

//------------------------------------------------------------------------------------------------------
// set alarm class parent of childs in the case of a parent or me=OFF or EOFF or STOP
IF me.AlarmConfig.bolChildrenAlarmPropagation THEN
	IF (CIf.Job.eParent_ActivAlmClass=E_AlmClass.EOFF) OR (CIf.Job.eParent_ActivAlmClass=E_AlmClass.OFF) OR (CIf.Job.eParent_ActivAlmClass=E_AlmClass.STOP) THEN
		SetAllChildAlmClass(CIf.Job.eParent_ActivAlmClass);
	ELSIF(CIf.Job.eMe_ActivAlmClass=E_AlmClass.EOFF) OR (CIf.Job.eMe_ActivAlmClass=E_AlmClass.OFF) OR (CIf.Job.eMe_ActivAlmClass=E_AlmClass.STOP) THEN
		SetAllChildAlmClass(CIf.Job.eMe_ActivAlmClass);
	ELSE
		// no important alarm for child active
		SetAllChildAlmClass(E_AlmClass.NONE);
	END_IF
END_IF
END_METHOD

METHOD PRIVATE CheckCmdValid : BOOL
VAR
	ii: UINT;
END_VAR
CheckCmdValid := FALSE;
FOR ii:=0 TO cMaxCmdPerCtrl BY 1 DO
	// check if a valid cmd
	IF (CIf.Job.aCmdList[ii].intCmd=cCMD_INITIALIZED) OR (CIf.Job.aCmdList[ii].intCmd=cCMD_DONE) THEN
		EXIT; // end for
	END_IF
	// check if a in this ctrl implemented cmd
	IF (CIf.Job.aCmdList[ii].intCmd=me.intCmd) THEN
		CheckCmdValid := TRUE;
	END_IF
END_FOR
END_METHOD

METHOD PROTECTED CheckParentAlmClass : BOOL
// --------------------------------------------------------------------------
// check alarm recation class of master													
// --------------------------------------------------------------------------
IF me.AlarmConfig.bolChildrenAlarmPropagation THEN
	IF (CIf.Job.eParent_ActivAlmClass = E_AlmClass.EOFF) THEN
		me.Alarm.eParent_ActivAlmClass := E_AlmClass.EOFF;
		// prevent automatic restart in manual or automatic
		IF (CIf.job.intACmd<>cCMD_PON) THEN // wait on startup until power on is ok
			CIf.job.intACmd := cCMD_DONE;
		END_IF
		
		IF (CIf.job.intMCmd<>cCMD_PON) THEN // wait on startup until power on is ok
			CIf.job.intMCmd := cCMD_DONE;
		END_IF
	ELSIF (CIf.Job.eParent_ActivAlmClass = E_AlmClass.OFF) THEN
		me.Alarm.eParent_ActivAlmClass := E_AlmClass.OFF;
	ELSIF (CIf.Job.eParent_ActivAlmClass = E_AlmClass.STOP) THEN
		me.Alarm.eParent_ActivAlmClass := E_AlmClass.STOP;
	ELSE
		me.Alarm.eParent_ActivAlmClass := E_AlmClass.NONE;
	END_IF
END_IF
END_METHOD

PROPERTY PUBLIC ChildrenAlarmPropagation : BOOL
GET
ChildrenAlarmPropagation := me.AlarmConfig.bolChildrenAlarmPropagation;
END_GET
SET
me.AlarmConfig.bolChildrenAlarmPropagation := ChildrenAlarmPropagation;
END_SET
END_PROPERTY

METHOD PUBLIC ClearAllSimulation : BOOL
VAR
	iIdx						: INT;
END_VAR
FOR iIdx := 0 TO UINT_TO_INT(Base_Const.cMaxNrOfChilds) DO
	IF CIf.Info.p_afbChild[iIdx] <> NULL THEN
		CIf.Info.p_afbChild[iIdx]^.ClearAllSimulation();
	END_IF
END_FOR

me.bolSimulateAllExecuted 	:= FALSE;
CIf.SwCfg.bolSimulation   	:= FALSE;
CIf.SwCfg.bolAllSimulation	:= FALSE;
END_METHOD

PROPERTY PUBLIC CtrlCIf : POINTER TO T_Ctrl_CIf
GET
CtrlCIf := ADR(CIf);
END_GET
END_PROPERTY

PROPERTY PUBLIC CtrlFB : POINTER TO FB_CtrlBASE
GET
CtrlFB := ADR(THIS^);
END_GET
END_PROPERTY

METHOD PUBLIC CtrlInit : BOOL
VAR
	udiTaskCnt: UDINT;
	fbGETCURTASKINDEX: Tc2_System.GETCURTASKINDEX;
END_VAR
IF (CIf.Info.bolInitDone=FALSE) THEN
	//automatic read out infos about FUB
	udiTaskCnt := TwinCAT_SystemInfoVarList._AppInfo.TaskCnt;
	fbGETCURTASKINDEX();
	udiTaskCnt := fbGETCURTASKINDEX.index;
	me.FUBInfo.udiSample_us := TwinCAT_SystemInfoVarList._TaskInfo[UDINT_TO_DINT(udiTaskCnt)].CycleTime/10; //[ms] X[100ns]/10 -> [us]
	me.FUBInfo.udiSample_ms := TwinCAT_SystemInfoVarList._TaskInfo[UDINT_TO_DINT(udiTaskCnt)].CycleTime/10000; //[ms] X[100ns]/10000 -> [ms]
	me.FUBInfo.bolCycleTimeBelowMS := me.FUBInfo.udiSample_us <= 1000;
	
	CIf.Info.bolInitDone  := TRUE;
END_IF
END_METHOD

METHOD PROTECTED CycleEndDuty : BOOL
me.eModeHistory := CIf.Job.eMode;				// save mode to detect mode switches
me.intCmdLast := me.intCmd;

// --------------------------------------------------------------------------
// switch to next State
// --------------------------------------------------------------------------
IF (me.StateMachine.intState<>me.StateMachine.intStateNext) THEN
	me.StateMachine.intState := me.StateMachine.intStateNext;  // set next state for next cycle
	IF (me.StateMachine.intState<>cSTA_SINGLE_ANSWER) THEN // only if no simulation is active
		CIf.Job.intState := me.StateMachine.intState;		// set information of actual state to controller interface
		CIf.Job.strState := THIS^.getCmdState(intCmdState:=CIf.Job.intState,bolState:=TRUE);
	ELSE
		CIf.Job.strState :=  TC2_STANDARD.CONCAT(STR1:='SINGLE_ANSWER-',STR2:=THIS^.getCmdState(intCmdState:=CIf.Job.intState,bolState:=TRUE));
	END_IF
	
	// delete SubState
	//me.SubStateMachine.intState := cSTA_DONE;
	//me.SubStateMachine.intStateNext := cSTA_DONE;
	
	// log state change
	me.stStateLogger.bolDoLog := TRUE;
	
	me.StateMachine.udiTimeInState_ms := 0; // reset timer
	me.StateMachine.udiTimeInState_us := 0; // reset timer
	me.SubStateMachine.udiTimeInState_ms := 0; // reset timer
	me.SubStateMachine.udiTimeInState_us := 0; // reset timer
	me.SubStateMachine.intState := cSTA_DONE;
	// log state change -> open point
ELSE
	// increment time in state	
	me.StateMachine.udiTimeInState_us := me.StateMachine.udiTimeInState_us + me.FUBInfo.udiSample_us;
	me.StateMachine.udiTimeInState_ms := me.StateMachine.udiTimeInState_ms + me.FUBInfo.udiSample_ms;
	me.StateMachine.relTimeInState_ms := UDINT_TO_REAL(me.StateMachine.udiTimeInState_us) / 1000.0;
END_IF


// --------------------------------------------------------------------------
// switch to next SubState
// --------------------------------------------------------------------------
IF (me.SubStateMachine.intState<>me.SubStateMachine.intStateNext) THEN
	me.SubStateMachine.intState := me.SubStateMachine.intStateNext;  // set next state for next cycle
	CIf.Job.strSubState := THIS^.getCmdState(intCmdState:=me.SubStateMachine.intState,bolState:=TRUE);
	me.SubStateMachine.udiTimeInState_ms := 0; // reset timer
	me.SubStateMachine.udiTimeInState_us := 0; // reset timer
	// log state change
	me.stStateLogger.bolDoLog := TRUE;
ELSE
	// increment time in state	
	me.SubStateMachine.udiTimeInState_us := me.SubStateMachine.udiTimeInState_us + me.FUBInfo.udiSample_us;
	me.SubStateMachine.udiTimeInState_ms := me.SubStateMachine.udiTimeInState_ms + me.FUBInfo.udiSample_ms;
	me.SubStateMachine.relTimeInState_ms := UDINT_TO_REAL(me.SubStateMachine.udiTimeInState_us) / 1000.0;
END_IF


// --------------------------------------------------------------------------
// entry state change in statelogger
// --------------------------------------------------------------------------
// access state logger system if enabled, central log pointer set and no handle allready received
IF ((CIf.SwCfg.bolEnStateLogger=TRUE) AND (me.stStateLogger.pfbBaseLog<>TC3_MEMMAN.NULL) AND (me.stStateLogger.pHandle=TC3_MEMMAN.NULL)) THEN
	// get handle for state logger
	me.stStateLogger.uinStatus_Handle := me.stStateLogger.pfbBaseLog^.M_GetHandle(Out_pHandle=>me.stStateLogger.pHandle );
END_IF

IF ((CIf.SwCfg.bolEnStateLogger=TRUE) AND (me.stStateLogger.pfbBaseLog<>TC3_MEMMAN.NULL) AND (me.stStateLogger.pHandle<>TC3_MEMMAN.NULL)) THEN
	IF (me.stStateLogger.bolDoLog=TRUE) THEN
		me.stStateLogger.strText1 := CIf.Info.strName;
		// concat string of state and sub statemachine
		IF (INT_TO_USINT(LEN(me.stStateLogger.strText1)+LEN(CIf.Job.strState) + 1 ) < BasLog.cMAX_CHAR_TEXT1) THEN
			me.stStateLogger.strText1 := CONCAT(me.stStateLogger.strText1, '#');
			me.stStateLogger.strText1 := CONCAT(me.stStateLogger.strText1, CIf.Job.strState);
			IF (INT_TO_USINT(LEN(me.stStateLogger.strText1)+LEN(CIf.Job.strSubState) + 1) < BasLog.cMAX_CHAR_TEXT1) THEN
				me.stStateLogger.strText1 := CONCAT(me.stStateLogger.strText1, '-');
				me.stStateLogger.strText1 := CONCAT(me.stStateLogger.strText1, CIf.Job.strSubState);
			END_IF
		END_IF
		// do entry in log queue
		me.stStateLogger.uinStatusWrite := me.stStateLogger.pfbBaseLog^.M_Log(In_pHandle:=me.stStateLogger.pHandle,In_udiLogType:=BasLog.cLOGTYPE_STATELOG,In_intCtrlID:=CIf.Info.intCtrlId,In_strText1:=me.stStateLogger.strText1,In_strText2:=me.stStateLogger.strText2,In_dinPar1:=me.StateMachine.intState,In_dinPar2:=me.SubStateMachine.intState,In_dinPar3:=me.stStateLogger.dinPar3,In_dinPar4:=me.stStateLogger.dinPar4) ;
		me.stStateLogger.bolDoLog := FALSE;
	END_IF
END_IF


// --------------------------------------------------------------------------
// Final state reached -> reset command
// --------------------------------------------------------------------------
IF (CIf.Job.intState=me.intCmd) THEN 
	CIf.Job.intACmd := cCMD_DONE;
	CIf.Job.intMCmd := cCMD_DONE;
END_IF


// --------------------------------------------------------------------------
// reset local alarm class
// --------------------------------------------------------------------------
IF (CIf.Job.bolAlmReset=TRUE) AND (CIf.Job.intState<>cSTA_ERROR) AND (CIf.Job.intState<>cSTA_ERRORQuit) THEN
	CIf.Job.eMe_ActivAlmClass := E_AlmClass.NONE;
	CIf.Job.bolAlmReset := FALSE;
END_IF


// --------------------------------------------------------------------------
// output bridge
// --------------------------------------------------------------------------
THIS^.IoOutBridge();	// digitale and analoge outputs or forcing write to hardware
END_METHOD

METHOD PROTECTED CycleStartDuty : BOOL

	// --------------------------------------------------------------------------
	// input bridge
	// --------------------------------------------------------------------------
	THIS^.IoInBridge(); // digitale and analoge inputs read from hardware or forcing

	// --------------------------------------------------------------------------
	// check alarm recation class of master													
	// --------------------------------------------------------------------------
	THIS^.CheckParentAlmClass();
	
	// ----------------------------------------------------------------------------------
	// check the highest active alarm -> set local class
	// ----------------------------------------------------------------------------------
	IF (me.Alarm.eParent_ActivAlmClass>CIf.job.eMe_ActivAlmClass) THEN
		me.Alarm.eActivAlmClass := me.Alarm.eParent_ActivAlmClass;
	ELSE
		me.Alarm.eActivAlmClass := CIf.job.eMe_ActivAlmClass;
	END_IF
	
	// ----------------------------------------------------------------------------------
	// check child me and set parent alarm class
	// ----------------------------------------------------------------------------------
	CheckChildAlmClass();
	
	// --------------------------------------------------------------------------
	// get command											
	// --------------------------------------------------------------------------
	IF (CIf.Job.eMode = E_Mode.MANU) THEN
		me.intCmd := CIf.Job.intMCmd;  
	ELSE
		IF (me.eModeHistory <> E_MODE.AUTO) THEN
			CIf.Job.intMCmd:= cCMD_DONE;	// reset manual command
			me.bolChangeBackToAUTO := TRUE;	// switch off  or .....
		END_IF
		CIf.Job.eMode := E_MODE.AUTO;
		me.intCmd := CIf.Job.intACmd;
	END_IF
	CIf.Job.strCmd := THIS^.getCmdState(intCmdState:=me.intCmd,bolState:=FALSE);
END_METHOD

METHOD PROTECTED EOFF_EntryAction : BOOL
VAR_INPUT
END_VAR
 // used for special events in EOFF
END_METHOD

PROPERTY PUBLIC EOffAlarmTransition : BOOL
GET
EOffAlarmTransition := NOT me.AlarmConfig.bolEOffAlarmTransitionDisable;
END_GET
SET
me.AlarmConfig.bolEOffAlarmTransitionDisable := NOT EOffAlarmTransition;
END_SET
END_PROPERTY

METHOD FB_init : BOOL
VAR_INPUT
	///if TRUE, the retain variables are initialized (warm start / cold start)
	bInitRetains: BOOL;
	///if TRUE, the instance afterwards gets moved into the copy code (online change)
	bInCopyCode: BOOL;
END_VAR
//------------------------------------------------------------------------------------------------------------------------
// enable cyclic call
me.bolActivate := TRUE;
// reset init flag
CIf.Info.bolInitDone := FALSE;

//------------------------------------------------------------------------------------------------------------------------
// to manually change in new FUB implementation!!!
// define valid commands for this controller
CIf.Job.aCmdList[0].intCmd := cCMD_PON;
CIf.Job.aCmdList[0].strName := 'Power On';
CIf.Job.aCmdList[0].bolAvailable := TRUE;

CIf.Job.aCmdList[1].intCmd := cCMD_OFF; // for test simulation single answer
CIf.Job.aCmdList[1].strName := 'OFF';
CIf.Job.aCmdList[1].bolAvailable := TRUE;

CIf.Job.aCmdList[2].intCmd := cCMD_EOFF;
CIf.Job.aCmdList[2].strName := 'Emergency OFF';
CIf.Job.aCmdList[2].bolAvailable := TRUE;

// set name of class/typ
CIf.Info.strType := 'FB_CtrlBase'; 

CIf.SwCfg.bolExist := TRUE;
CIf.SwCfg.bolSimulation := FALSE;
CIf.SwCfg.bolEnStateLogger := TRUE;

//------------------------------------------------------------------------------------------------------------------------
CIf.Info.strName := getStrInstanceName(strMyInstancePath); // get name of instance
CIf.Info.strInstancePath := strMyInstancePath;
CIf.Info.uinChildNbr := 0;
me.bolSimulateAllExecuted := FALSE;
me.AlarmConfig.bolEOffAlarmTransitionDisable := FALSE;
me.AlarmConfig.bolEOffCmdTransitionDisable := FALSE;
me.AlarmConfig.bolOffAlarmTransitionDisable := FALSE;
me.AlarmConfig.bolOffCmdTransitionDisable := FALSE;
me.AlarmConfig.bolChildrenAlarmPropagation := TRUE;
END_METHOD

METHOD PROTECTED FurtherReactions : BOOL
;

// Example Implementation
(*
IF (	(NOT me.AlarmConfig.bolOffAlarmTransitionDisable)	AND (me.Alarm.eActivAlmClass=E_AlmClass.STOP)
	AND (me.StateMachine.intState<>cSTA_ERROR)				AND	(me.StateMachine.intState<>cSTA_ERRORQuit)
	AND	(me.StateMachine.intState<>cSTA_EOFF)				AND	(me.StateMachine.intState<>cSTA_EOFFBusy)
	AND	(me.StateMachine.intState<>cSTA_OFF)				AND	(me.StateMachine.intState<>cSTA_OFFBusy)
	AND (me.StateMachine.intState<>cSTA_STOP)				AND (me.StateMachine.intState<>cSTA_STOPBusy)
	AND	(me.StateMachine.intState>cSTA_PON)) THEN
	
	me.StateMachine.intStateNext := cSTA_STOPBusy;
	me.StateMachine.intState := cSTA_DONE;
	
ELSIF (	(NOT me.AlarmConfig.bolOffAlarmTransitionDisable)	AND (me.Alarm.eActivAlmClass=E_AlmClass.TSTOP)
	AND (me.StateMachine.intState<>cSTA_ERROR)				AND	(me.StateMachine.intState<>cSTA_ERRORQuit)
	AND	(me.StateMachine.intState<>cSTA_EOFF)				AND	(me.StateMachine.intState<>cSTA_EOFFBusy)
	AND	(me.StateMachine.intState<>cSTA_OFF)				AND	(me.StateMachine.intState<>cSTA_OFFBusy)
	AND (me.StateMachine.intState<>cSTA_STOP)				AND (me.StateMachine.intState<>cSTA_STOPBusy)
	AND	(me.StateMachine.intState>cSTA_PON)) THEN
	
	me.StateMachine.intStateNext := cSTA_STOPBusy;
	me.StateMachine.intState := cSTA_DONE;
	
END_IF
*)
END_METHOD

METHOD PROTECTED getCmdState : STRING
VAR_INPUT
	intCmdState: INT;
	bolState: BOOL;
END_VAR
// get string cmd/state string information in runtime
IF (bolState=FALSE) THEN
	// cmd's
	CASE intCmdState OF
		cCMD_DONE: 
			getCmdState := 'cCMD_DONE';
		cCMD_INITIALIZED: 
			getCmdState := 'cCMD_INITIALIZED';
		cCMD_PON: 
			getCmdState := 'cCMD_PON';
		cCMD_EOFF: 
			getCmdState := 'cCMD_EOFF';
		cCMD_OFF: 
			getCmdState := 'cCMD_OFF';
		cCMD_INIT: 
			getCmdState := 'cCMD_INIT';
		cCMD_RUN: 
			getCmdState := 'cCMD_RUN';
		cCMD_STOP: 
			getCmdState := 'cCMD_STOP';
		cCMD_TSTOP: 
			getCmdState := 'cCMD_TSTOP';
	END_CASE;
ELSE
	// states
	CASE intCmdState OF
		cSTA_DONE: 
			getCmdState := 'cSTA_DONE';
		cSTA_INITIALIZED: 
			getCmdState := 'cSTA_INITIALIZED';
		cSTA_PONBusy: 
			getCmdState := 'cSTA_PONBusy';
		cSTA_PON: 
			getCmdState := 'cSTA_PON';
		cSTA_EOFFBusy: 
			getCmdState := 'cSTA_EOFFBusy';
		cSTA_EOFF: 
			getCmdState := 'cSTA_EOFF';
		cSTA_OFFBusy: 
			getCmdState := 'cSTA_OFFBusy';
		cSTA_OFF: 
			getCmdState := 'cSTA_OFF';
		cSTA_INITBusy: 
			getCmdState := 'cSTA_INITBusy';
		cSTA_INIT: 
			getCmdState := 'cSTA_INIT';
		cSTA_RUNBusy: 
			getCmdState := 'cSTA_RUNBusy';
		cSTA_RUN: 
			getCmdState := 'cSTA_RUN';
		cSTA_STOPBusy: 
			getCmdState := 'cSTA_STOPBusy';
		cSTA_STOP: 
			getCmdState := 'cSTA_STOP';
		cSTA_TSTOPBusy: 
			getCmdState := 'cSTA_TSTOPBusy';
		cSTA_TSTOP: 
			getCmdState := 'cSTA_TSTOP';
		cSTA_ERROR: 
			getCmdState := 'cSTA_ERROR';
		cSTA_ERRORQuit: 
			getCmdState := 'cSTA_ERRORQuit';
		cSTA_SINGLE_ANSWER: 
			getCmdState := 'cSTA_SINGLE_ANSWER';
	END_CASE;
END_IF
END_METHOD

METHOD PUBLIC iniAllCtrlArrays : BOOL
VAR_INPUT
	p_pCtrlFbBaseArray	: POINTER TO POINTER TO FB_CtrlBase;
	p_pCtrlCIfArray		: POINTER TO POINTER TO T_Ctrl_CIf;
	intCtrlID		: INT;
END_VAR
iniAllCtrlArrays := FALSE;

IF (TRUE) THEN//e_CtrlID <= E_CtrlId.E_CtrlIdMax) THEN
	p_pCtrlFbBaseArray[intCtrlID] 	:= THIS;
	THIS^.CIf.Info.intCtrlID := intCtrlID;
	p_pCtrlCIfArray[intCtrlID] := CtrlCIf;
	iniAllCtrlArrays := TRUE;
END_IF
END_METHOD

PROPERTY PUBLIC InstancePath : STRING
GET
InstancePath := strMyInstancePath;
END_GET
END_PROPERTY

METHOD PROTECTED IoInBridge : BOOL
// digitale and analoge inputs read from hardware or forcing
IF (CIf.SwCfg.bolSimulation = FALSE) THEN
	//KVO??? alternative only without feedback getIn(ctrl.ifc.Job.bol_Force ,ADR(ctrl.In.bol_PosSwitchBasicDefTyp);
	//ctrl.In.bol_PosSwitchBasicDefTyp.intern := getIn(ctrl.ifc.Job.bol_Force ,ADR(ctrl.In.bol_PosSwitchBasicDefTyp);
ELSE
	//simulation of global IO
END_IF
END_METHOD

METHOD PROTECTED IoOutBridge : BOOL
// digitale and analoge inputs read from hardware or forcing
IF (CIf.SwCfg.bolSimulation = FALSE) THEN


//KVO??? alternative only without feedback getIn(ctrl.ifc.Job.bol_Force ,ADR(ctrl.In.bol_PosSwitchBasicDefTyp);
	// check interlocks to prevent damages
	//IF (SIf.Ilk.bolOverwrite=FALSE) THEN
		//IF (SIf.Ilk.bolOut=FALSE) THEN
			//ctrl.Out.bolOut.map := setOut(ctrl.ifc.Job.bol_Force ,ADR(ctrl.Out.bolOut);
		//ELSE
			// switch off???
			// error??
		//END_IF
	//end_if

	//THIS^.Out_bolOut := SIf.Out.bolOut.map;

END_IF
END_METHOD

PROPERTY PUBLIC OffAlarmTransition : BOOL
GET
OffAlarmTransition := NOT me.AlarmConfig.bolOffAlarmTransitionDisable;
END_GET
SET
me.AlarmConfig.bolOffAlarmTransitionDisable := NOT OffAlarmTransition;
END_SET
END_PROPERTY

METHOD PROTECTED ResetSubState : BOOL
VAR_INPUT
	In_FirstState : INT; // first state to start with
END_VAR
// reset the substate variables and set first state
me.SubStateMachine.intStateHistory := 0;
me.SubStateMachine.intStateLastCycle := 0;
me.SubStateMachine.intStateNext := In_FirstState;
me.SubStateMachine.intState := me.SubStateMachine.intStateNext -1; // -> change state at the end -> log state change possibel
END_METHOD

METHOD PROTECTED SetAllChildAlmClass : BOOL
VAR_INPUT
	In_intSetAlmClass : INT;
END_VAR
VAR
	uinIdx: UINT;
END_VAR
IF (CIf.Info.uinChildNbr > 0) THEN
	FOR uinIdx := 0 TO CIf.Info.uinChildNbr - 1 DO
		CIf.Info.p_aCIf[uinIdx]^.Job.eParent_ActivAlmClass := In_intSetAlmClass;
	END_FOR
END_IF
END_METHOD

METHOD PROTECTED SetAllChildCmd
VAR_INPUT
	In_intSetAcmd : INT;
END_VAR
VAR
	uinIdx: UINT;
END_VAR
IF (CIf.Info.uinChildNbr > 0) THEN
	FOR uinIdx := 0 TO CIf.Info.uinChildNbr - 1 DO
		CIf.Info.p_aCIf[uinIdx]^.Job.intACmd := In_intSetAcmd;
	END_FOR
END_IF
END_METHOD

METHOD PUBLIC SetAllSimulation : BOOL
VAR
	iIdx						: INT;
END_VAR
FOR iIdx := 0 TO UINT_TO_INT(Base_Const.cMaxNrOfChilds) DO
	IF CIf.Info.p_afbChild[iIdx] <> NULL THEN
		CIf.Info.p_afbChild[iIdx]^.SetAllSimulation();
	END_IF
END_FOR

me.bolSimulateAllExecuted := TRUE;
CIf.SwCfg.bolSimulation   := TRUE;
CIf.SwCfg.bolAllSimulation	:= TRUE;
END_METHOD

METHOD PROTECTED sta_EOFF : BOOL
// state implemetation
//--------------------------------------------------------------------------------------
// Entry action
	IF (me.StateMachine.intState<>me.StateMachine.intStateLastCycle) THEN
		me.StateMachine.intStateLastCycle := me.StateMachine.intState;
	END_IF


//--------------------------------------------------------------------------------------
// Cyclic action
	IF (me.StateMachine.intState=me.StateMachine.intStateLastCycle) THEN
		
		// State Change Condition
		IF (me.Alarm.eActivAlmClass<>E_AlmClass.EOFF) AND (me.intCmd<>cCMD_EOFF) AND (me.intCmd<>cCMD_DONE) THEN
			IF (TRUE) THEN
				me.StateMachine.intStateNext := cSTA_OFFBusy;
			END_IF
		END_IF
		
	END_IF


//--------------------------------------------------------------------------------------
// Exit action
	IF (me.StateMachine.intState<>me.StateMachine.intStateNext) THEN
		;
	END_IF
END_METHOD

METHOD PROTECTED sta_EOFFBusy : BOOL
VAR_INPUT
END_VAR
// state implemetation
//--------------------------------------------------------------------------------------
// Entry action
	IF (me.StateMachine.intState<>me.StateMachine.intStateLastCycle) THEN
		me.StateMachine.intStateLastCycle := me.StateMachine.intState;
		EOFF_EntryAction(); // used for special events in EOFF
		// Set commandos not only in entry action because of possible errors or manual/auto changes
		// PRE/AVME 06.01.2014
		//SetAllChildCmd(cCMD_EOFF); // set acmd off all childs 
	END_IF


//--------------------------------------------------------------------------------------
// Cyclic action
	IF (me.StateMachine.intState=me.StateMachine.intStateLastCycle) THEN
		
		SetAllChildCmd(cCMD_EOFF); // set acmd off all childs 
	
		// check if all childs have reached the state
		IF CheckAllChildState(cSTA_EOFF) THEN
			me.StateMachine.intStateNext := cSTA_EOFF;
		END_IF
	END_IF


//--------------------------------------------------------------------------------------
// Exit action
	IF (me.StateMachine.intState<>me.StateMachine.intStateNext) THEN
		;
	END_IF
END_METHOD

METHOD PROTECTED sta_ERROR : BOOL
// state implemetation
//--------------------------------------------------------------------------------------
// Entry action
	IF (me.StateMachine.intState<>me.StateMachine.intStateLastCycle) THEN
		me.StateMachine.intStateHistory := me.StateMachine.intStateLastCycle; // -> possibillity to go back to state before error
		me.StateMachine.intStateLastCycle := me.StateMachine.intState;
		
	END_IF


//--------------------------------------------------------------------------------------
// Cyclic action
	IF (me.StateMachine.intState=me.StateMachine.intStateLastCycle) THEN
		
		;
		
		
		// State Change Condition
		IF (CIf.Job.bolAlmReset = TRUE) THEN
			me.StateMachine.intStateNext := cSTA_ERRORQuit;
		END_IF
	END_IF




//--------------------------------------------------------------------------------------
// Exit action
	IF (me.StateMachine.intState<>me.StateMachine.intStateNext) THEN
		;
	END_IF
END_METHOD

METHOD PROTECTED sta_ERRORQuit : BOOL
// state implemetation
//--------------------------------------------------------------------------------------
// Entry action
	IF (me.StateMachine.intState<>me.StateMachine.intStateLastCycle) THEN
		me.StateMachine.intStateLastCycle := me.StateMachine.intState;
	END_IF


//--------------------------------------------------------------------------------------
// Cyclic action
	IF (me.StateMachine.intState=me.StateMachine.intStateLastCycle) THEN
		
		CIf.Job.eMe_ActivAlmClass := E_AlmClass.NONE; // reset feedback channel for parent
		CIf.Job.bolAlmReset := FALSE;
		
		// State Change Condition
		IF (me.StateMachine.intStateHistory<=cSTA_PON) THEN
			me.StateMachine.intStateNext := cSTA_PONBusy;
		ELSE
			me.StateMachine.intStateNext := cSTA_OFFBusy;
		END_IF
		
	END_IF


//--------------------------------------------------------------------------------------
// Exit action
	IF (me.StateMachine.intState<>me.StateMachine.intStateNext) THEN
		;
	END_IF
END_METHOD

METHOD PROTECTED sta_OFF : BOOL
// state implemetation
//--------------------------------------------------------------------------------------
// Entry action
	IF (me.StateMachine.intState<>me.StateMachine.intStateLastCycle) THEN
		me.StateMachine.intStateLastCycle := me.StateMachine.intState;
		
	END_IF


//--------------------------------------------------------------------------------------
// Cyclic action
	IF (me.StateMachine.intState=me.StateMachine.intStateLastCycle) THEN
		
		;
		
		
		// State Change Condition
		IF ((me.Alarm.eActivAlmClass<>E_AlmClass.EOFF) AND (me.Alarm.eActivAlmClass<>E_AlmClass.OFF)) THEN
			IF (TRUE) THEN
				;	//me.StateMachine.intStateNext := cSTA_PON;
			END_IF
		END_IF;
	END_IF




//--------------------------------------------------------------------------------------
// Exit action
	IF (me.StateMachine.intState<>me.StateMachine.intStateNext) THEN
		;
	END_IF
END_METHOD

METHOD PROTECTED sta_OFFBusy : BOOL
// state implemetation
//--------------------------------------------------------------------------------------
// Entry action
	IF (me.StateMachine.intState<>me.StateMachine.intStateLastCycle) THEN
		me.StateMachine.intStateLastCycle := me.StateMachine.intState;
		
		// Set commandos not only in entry action because of possible errors or manual/auto changes
		// PRE/AVME 06.01.2014
		//SetAllChildCmd(cCMD_OFF); // set acmd off all childs 
	END_IF


//--------------------------------------------------------------------------------------
// Cyclic action
	IF (me.StateMachine.intState=me.StateMachine.intStateLastCycle) THEN
		
		SetAllChildCmd(cCMD_OFF); // set acmd off all childs 
		
		// State Change Condition
		IF (CheckAllChildState(cSTA_OFF)) THEN
			me.StateMachine.intStateNext := cSTA_OFF;
		END_IF
	END_IF




//--------------------------------------------------------------------------------------
// Exit action
	IF (me.StateMachine.intState<>me.StateMachine.intStateNext) THEN
		;
	END_IF
END_METHOD

METHOD PROTECTED sta_PON : BOOL
// state implemetation
//--------------------------------------------------------------------------------------
// Entry action
	IF (me.StateMachine.intState<>me.StateMachine.intStateLastCycle) THEN
		me.StateMachine.intStateLastCycle := me.StateMachine.intState;
		
	END_IF


//--------------------------------------------------------------------------------------
// Cyclic action
	IF (me.StateMachine.intState=me.StateMachine.intStateLastCycle) THEN
		
		;
		
		
		// State Change Condition
		IF (me.intCmd<>cCMD_PON) AND (me.intCmd<>cCMD_DONE) THEN
			me.StateMachine.intStateNext := cSTA_EOFFBusy;
		END_IF
	END_IF




//--------------------------------------------------------------------------------------
// Exit action
	IF (me.StateMachine.intState<>me.StateMachine.intStateNext) THEN
		;
	END_IF
END_METHOD

METHOD PROTECTED sta_PONBusy : BOOL
// state implemetation
//--------------------------------------------------------------------------------------
// Entry action
	IF (me.StateMachine.intState<>me.StateMachine.intStateLastCycle) THEN
		me.StateMachine.intStateLastCycle := me.StateMachine.intState;
		
		SetAllChildCmd(cCMD_PON); // set acmd off all childs 
	END_IF


//--------------------------------------------------------------------------------------
// Cyclic action
	IF (me.StateMachine.intState=me.StateMachine.intStateLastCycle) THEN
		
		;
		
		
		// State Change Condition
		IF CheckAllChildState(cSTA_PON) THEN
			me.StateMachine.intStateNext := cSTA_PON;
		END_IF
	END_IF




//--------------------------------------------------------------------------------------
// Exit action
	IF (me.StateMachine.intState<>me.StateMachine.intStateNext) THEN
		;
	END_IF
END_METHOD

METHOD PROTECTED sta_SINGLE_ANSWER : BOOL
// state implemetation of SINGLE_ANSWER
//--------------------------------------------------------------------------------------
// Entry action
	IF (me.StateMachine.intState<>me.StateMachine.intStateLastCycle) THEN
		me.StateMachine.intStateLastCycle := me.StateMachine.intState;
		
	END_IF


//--------------------------------------------------------------------------------------
// Cyclic action
	IF (me.StateMachine.intState=me.StateMachine.intStateLastCycle) THEN
		
		// Reset pending alarm class
		CIf.Job.eMe_ActivAlmClass := E_AlmClass.NONE;
	
		IF ((me.intCmd<>cCMD_INITIALIZED) AND (me.intCmd<>cCMD_DONE)) THEN
			IF (THIS^.CheckCmdValid()=TRUE) THEN
				IF (me.intCmd<>me.intCmdLast) THEN
					me.StateMachine.udiTimeInState_ms := 0;  // reset timer
				END_IF
				IF (me.StateMachine.udiTimeInState_ms >= me.StateMachine.udiStateSimSetTime_ms) THEN
					CIf.Job.intState := me.intCmd; // simulate final state
				ELSE
					CIf.Job.intState := me.intCmd-1; // simulate busy state
				END_IF
			END_IF
		END_IF
		
		// State Change Condition
		IF (FALSE) THEN
			;
		ELSIF (CIf.SwCfg.bolExist=TRUE) THEN
			me.StateMachine.intStateNext := cSTA_PONBusy;
		END_IF
	END_IF




//--------------------------------------------------------------------------------------
// Exit action
	IF (me.StateMachine.intState<>me.StateMachine.intStateNext) THEN
		;
	END_IF
END_METHOD

METHOD PROTECTED StateMachine : BOOL

